Yaskawa INFORM job: DEMO_ROOF_SIDE_0625_3PAINT_57.JBI

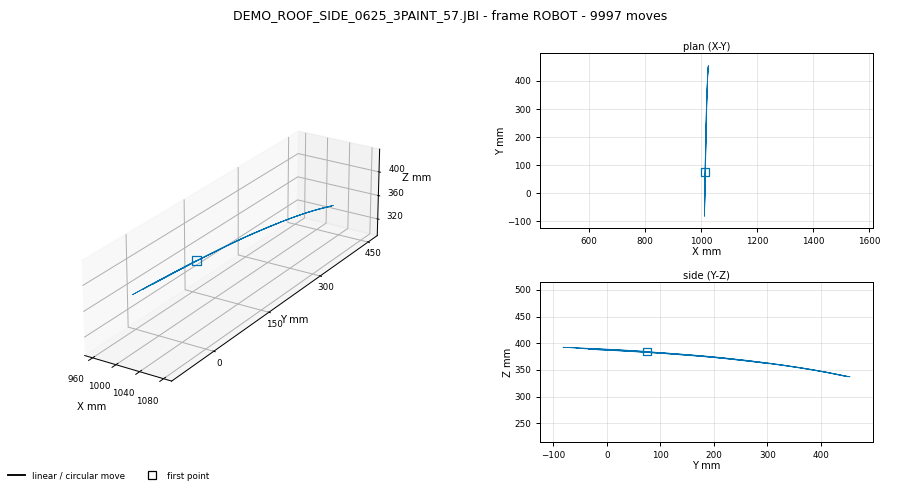
[picture p0: tool path of DEMO_ROOF_SIDE_0625_3PAINT_57.JBI in frame ROBOT, 9997 of 9997 moves have a stored position in this frame; points joined in program order, loops and branches not executed]
/JOB
//NAME DEMO_ROOF_SIDE_0625_3PAINT57
//POS
///NPOS 9997,0,0,0,0,0
///TOOL 0
///USER 0
///POSTYPE ROBOT
///RECTAN
///RCONF 1,0,0,0,0,0,0,0,0,0,0,0,0,0,0,0,0,0,0,0,0,0,0,0
C00000=1015.921,75.710,384.669,166.381,56.145,160.225
C00001=1015.916,75.460,384.686,166.378,56.154,160.227
C00002=1015.911,75.211,384.702,166.376,56.164,160.228
C00003=1015.906,74.930,384.720,166.373,56.174,160.229
C00004=1015.900,74.649,384.737,166.370,56.185,160.231
C00005=1015.894,74.368,384.755,166.367,56.195,160.232
C00006=1015.889,74.087,384.774,166.365,56.207,160.234
C00007=1015.884,73.838,384.789,166.362,56.215,160.235
C00008=1015.879,73.587,384.805,166.358,56.225,160.236
C00009=1015.874,73.339,384.822,166.356,56.235,160.237
C00010=1015.869,73.089,384.837,166.353,56.244,160.238
C00011=1015.864,72.840,384.854,166.351,56.253,160.240
C00012=1015.859,72.590,384.869,166.348,56.263,160.241
C00013=1015.855,72.341,384.885,166.346,56.272,160.242
C00014=1015.849,72.091,384.902,166.344,56.282,160.243
C00015=1015.844,71.842,384.917,166.341,56.291,160.245
C00016=1015.840,71.593,384.933,166.339,56.301,160.246
C00017=1015.834,71.343,384.949,166.336,56.310,160.247
C00018=1015.830,71.093,384.965,166.334,56.319,160.248
C00019=1015.825,70.844,384.981,166.332,56.329,160.250
C00020=1015.820,70.594,384.997,166.328,56.339,160.251
C00021=1015.815,70.345,385.012,166.326,56.348,160.252
C00022=1015.810,70.096,385.028,166.323,56.357,160.253
C00023=1015.806,69.847,385.044,166.320,56.366,160.254
C00024=1015.800,69.597,385.060,166.318,56.376,160.256
C00025=1015.795,69.348,385.076,166.316,56.385,160.257
C00026=1015.790,69.098,385.091,166.313,56.395,160.258
C00027=1015.785,68.848,385.107,166.311,56.404,160.259
C00028=1015.781,68.599,385.124,166.308,56.414,160.261
C00029=1015.776,68.350,385.139,166.306,56.423,160.262
C00030=1015.771,68.100,385.155,166.303,56.432,160.263
C00031=1015.766,67.850,385.170,166.301,56.441,160.264
C00032=1015.761,67.601,385.187,166.298,56.451,160.266
C00033=1015.756,67.352,385.202,166.296,56.460,160.267
C00034=1015.751,67.103,385.217,166.294,56.469,160.268
C00035=1015.746,66.853,385.233,166.290,56.479,160.269
C00036=1015.741,66.603,385.248,166.288,56.489,160.271
C00037=1015.737,66.354,385.264,166.285,56.498,160.272
C00038=1015.731,66.105,385.280,166.283,56.508,160.273
C00039=1015.726,65.855,385.296,166.280,56.516,160.274
C00040=1015.721,65.606,385.311,166.278,56.526,160.275
C00041=1015.716,65.356,385.327,166.275,56.535,160.277
C00042=1015.712,65.107,385.342,166.273,56.545,160.278
C00043=1015.706,64.857,385.358,166.271,56.554,160.279
C00044=1015.701,64.607,385.373,166.268,56.564,160.281
C00045=1015.697,64.359,385.390,166.266,56.573,160.282
C00046=1015.692,64.109,385.405,166.263,56.582,160.283
C00047=1015.686,63.859,385.420,166.261,56.591,160.284
C00048=1015.682,63.610,385.436,166.258,56.601,160.285
C00049=1015.677,63.360,385.451,166.256,56.610,160.287
C00050=1015.672,63.111,385.466,166.253,56.620,160.288
C00051=1015.667,62.862,385.482,166.250,56.630,160.289
C00052=1015.662,62.612,385.498,166.248,56.639,160.290
C00053=1015.657,62.362,385.513,166.245,56.648,160.291
C00054=1015.652,62.113,385.528,166.243,56.658,160.293
C00055=1015.647,61.864,385.543,166.241,56.667,160.294
C00056=1015.642,61.615,385.558,166.238,56.676,160.295
C00057=1015.636,61.364,385.573,166.236,56.686,160.297
C00058=1015.631,61.115,385.588,166.233,56.696,160.298
C00059=1015.626,60.865,385.604,166.230,56.705,160.299
C00060=1015.622,60.616,385.619,166.228,56.715,160.300
C00061=1015.617,60.367,385.635,166.226,56.724,160.302
C00062=1015.611,60.117,385.650,166.223,56.734,160.303
C00063=1015.606,59.867,385.665,166.221,56.743,160.304
C00064=1015.601,59.617,385.680,166.218,56.753,160.305
C00065=1015.596,59.368,385.695,166.215,56.763,160.307
C00066=1015.591,59.119,385.710,166.213,56.772,160.308
C00067=1015.585,58.826,385.728,166.210,56.783,160.309
C00068=1015.579,58.533,385.745,166.207,56.795,160.311
C00069=1015.573,58.240,385.763,166.204,56.805,160.312
C00070=1015.567,57.947,385.782,166.201,56.816,160.314
C00071=1015.563,57.697,385.796,166.199,56.826,160.315
C00072=1015.558,57.447,385.811,166.197,56.835,160.316
C00073=1015.553,57.198,385.826,166.194,56.845,160.317
C00074=1015.547,56.949,385.842,166.191,56.854,160.319
C00075=1015.542,56.700,385.857,166.189,56.864,160.320
C00076=1015.538,56.450,385.871,166.186,56.873,160.321
C00077=1015.533,56.201,385.886,166.184,56.882,160.322
C00078=1015.527,55.951,385.902,166.182,56.892,160.324
C00079=1015.522,55.701,385.917,166.179,56.901,160.325
C00080=1015.517,55.451,385.932,166.177,56.911,160.326
C00081=1015.512,55.202,385.947,166.174,56.920,160.327
C00082=1015.507,54.953,385.962,166.172,56.929,160.328
C00083=1015.503,54.710,385.976,166.170,56.939,160.330
C00084=1015.498,54.466,385.991,166.167,56.948,160.331
C00085=1015.493,54.222,386.006,166.165,56.957,160.332
C00086=1015.488,53.979,386.021,166.162,56.966,160.333
C00087=1015.483,53.735,386.035,166.160,56.975,160.334
C00088=1015.478,53.492,386.050,166.158,56.984,160.336
C00089=1015.473,53.248,386.064,166.156,56.993,160.337
C00090=1015.468,53.004,386.079,166.153,57.002,160.338
C00091=1015.463,52.755,386.094,166.150,57.012,160.339
C00092=1015.458,52.506,386.109,166.148,57.021,160.341
C00093=1015.453,52.256,386.124,166.145,57.030,160.342
C00094=1015.448,52.007,386.139,166.143,57.039,160.343
C00095=1015.443,51.757,386.154,166.141,57.049,160.344
C00096=1015.439,51.508,386.168,166.138,57.058,160.345
C00097=1015.434,51.258,386.184,166.136,57.067,160.347
C00098=1015.428,51.009,386.199,166.134,57.077,160.348
C00099=1015.424,50.759,386.213,166.131,57.086,160.349
C00100=1015.419,50.510,386.228,166.129,57.095,160.350
C00101=1015.414,50.261,386.244,166.126,57.104,160.351
C00102=1015.409,50.011,386.258,166.124,57.114,160.353
C00103=1015.404,49.761,386.273,166.121,57.123,160.354
C00104=1015.399,49.512,386.288,166.119,57.132,160.355
C00105=1015.394,49.262,386.303,166.116,57.142,160.356
C00106=1015.389,49.013,386.318,166.114,57.150,160.357
C00107=1015.384,48.763,386.333,166.112,57.160,160.359
C00108=1015.379,48.514,386.348,166.109,57.169,160.360
C00109=1015.374,48.265,386.363,166.107,57.178,160.361
C00110=1015.369,48.015,386.377,166.104,57.187,160.362
C00111=1015.364,47.766,386.393,166.102,57.197,160.363
C00112=1015.360,47.515,386.408,166.099,57.206,160.364
C00113=1015.355,47.266,386.423,166.098,57.215,160.366
C00114=1015.351,47.016,386.437,166.095,57.224,160.367
C00115=1015.346,46.767,386.452,166.093,57.233,160.368
C00116=1015.341,46.518,386.468,166.090,57.242,160.369
C00117=1015.336,46.268,386.482,166.088,57.252,160.370
C00118=1015.331,46.019,386.497,166.085,57.260,160.371
C00119=1015.327,45.769,386.511,166.083,57.270,160.373
C00120=1015.322,45.520,386.526,166.080,57.279,160.374
C00121=1015.317,45.270,386.541,166.077,57.288,160.375
C00122=1015.312,45.021,386.556,166.075,57.297,160.376
C00123=1015.307,44.771,386.571,166.073,57.306,160.377
C00124=1015.302,44.522,386.586,166.071,57.315,160.379
C00125=1015.297,44.272,386.600,166.069,57.324,160.380
C00126=1015.292,44.023,386.615,166.066,57.333,160.381
C00127=1015.288,43.773,386.630,166.064,57.342,160.382
C00128=1015.282,43.523,386.645,166.061,57.351,160.383
C00129=1015.278,43.274,386.659,166.058,57.360,160.384
C00130=1015.273,43.025,386.674,166.057,57.369,160.386
C00131=1015.267,42.744,386.691,166.054,57.379,160.387
C00132=1015.262,42.463,386.707,166.051,57.389,160.388
C00133=1015.257,42.181,386.724,166.049,57.400,160.390
C00134=1015.251,41.900,386.740,166.046,57.410,160.391
C00135=1015.246,41.651,386.755,166.044,57.419,160.392
C00136=1015.241,41.401,386.770,166.041,57.428,160.393
C00137=1015.236,41.151,386.784,166.039,57.438,160.394
C00138=1015.231,40.902,386.799,166.036,57.447,160.395
C00139=1015.227,40.653,386.813,166.034,57.456,160.397
C00140=1015.221,40.403,386.827,166.031,57.465,160.398
C00141=1015.217,40.153,386.841,166.029,57.474,160.399
C00142=1015.212,39.904,386.856,166.026,57.484,160.400
C00143=1015.207,39.654,386.871,166.024,57.492,160.401
C00144=1015.201,39.405,386.885,166.022,57.502,160.403
C00145=1015.197,39.155,386.899,166.019,57.511,160.404
C00146=1015.192,38.906,386.914,166.017,57.519,160.405
C00147=1015.187,38.657,386.928,166.015,57.529,160.406
C00148=1015.182,38.407,386.942,166.012,57.538,160.407
C00149=1015.177,38.157,386.957,166.010,57.548,160.409
C00150=1015.172,37.908,386.972,166.008,57.556,160.410
C00151=1015.167,37.658,386.986,166.005,57.565,160.411
C00152=1015.163,37.409,387.000,166.003,57.575,160.412
C00153=1015.158,37.159,387.014,166.000,57.584,160.413
C00154=1015.152,36.909,387.028,165.999,57.592,160.414
C00155=1015.147,36.660,387.043,165.996,57.601,160.415
C00156=1015.143,36.410,387.058,165.994,57.611,160.417
C00157=1015.137,36.161,387.072,165.991,57.620,160.418
C00158=1015.133,35.911,387.086,165.989,57.629,160.419
C00159=1015.127,35.662,387.100,165.986,57.638,160.420
C00160=1015.123,35.412,387.114,165.984,57.647,160.421
C00161=1015.117,35.162,387.128,165.982,57.657,160.423
C00162=1015.113,34.913,387.142,165.979,57.666,160.424
C00163=1015.108,34.664,387.156,165.977,57.675,160.425
C00164=1015.103,34.414,387.170,165.974,57.684,160.426
C00165=1015.097,34.164,387.184,165.971,57.693,160.427
C00166=1015.093,33.914,387.199,165.969,57.703,160.428
C00167=1015.088,33.665,387.212,165.967,57.712,160.429
C00168=1015.083,33.416,387.227,165.964,57.720,160.430
C00169=1015.078,33.166,387.240,165.963,57.730,160.432
C00170=1015.073,32.916,387.255,165.960,57.739,160.433
C00171=1015.068,32.667,387.268,165.958,57.747,160.434
C00172=1015.063,32.418,387.282,165.956,57.757,160.435
C00173=1015.058,32.168,387.297,165.953,57.766,160.436
C00174=1015.052,31.918,387.311,165.950,57.775,160.438
C00175=1015.048,31.669,387.325,165.948,57.785,160.439
C00176=1015.043,31.419,387.339,165.946,57.794,160.440
C00177=1015.038,31.170,387.353,165.943,57.802,160.441
C00178=1015.033,30.921,387.367,165.941,57.811,160.442
C00179=1015.028,30.671,387.381,165.939,57.820,160.443
C00180=1015.023,30.421,387.395,165.937,57.829,160.445
C00181=1015.018,30.171,387.409,165.934,57.838,160.446
C00182=1015.014,29.922,387.422,165.931,57.847,160.447
C00183=1015.008,29.672,387.436,165.929,57.856,160.448
C00184=1015.003,29.422,387.450,165.926,57.865,160.449
C00185=1014.998,29.174,387.464,165.925,57.874,160.450
C00186=1014.994,28.924,387.478,165.923,57.883,160.451
C00187=1014.988,28.674,387.492,165.920,57.892,160.453
C00188=1014.984,28.425,387.506,165.917,57.901,160.454
C00189=1014.979,28.175,387.520,165.915,57.910,160.455
C00190=1014.974,27.925,387.535,165.913,57.919,160.456
C00191=1014.969,27.676,387.547,165.911,57.928,160.457
C00192=1014.965,27.426,387.562,165.909,57.937,160.458
C00193=1014.959,27.176,387.576,165.906,57.946,160.459
C00194=1014.954,26.928,387.589,165.903,57.955,160.460
C00195=1014.949,26.646,387.605,165.901,57.965,160.462
C00196=1014.943,26.366,387.620,165.898,57.975,160.463
C00197=1014.937,26.085,387.635,165.895,57.985,160.464
C00198=1014.932,25.804,387.651,165.893,57.996,160.466
C00199=1014.927,25.554,387.664,165.891,58.004,160.467
C00200=1014.922,25.304,387.679,165.889,58.013,160.468
C00201=1014.917,25.055,387.692,165.886,58.022,160.469
C00202=1014.912,24.805,387.706,165.883,58.031,160.470
C00203=1014.906,24.555,387.719,165.881,58.040,160.471
C00204=1014.902,24.306,387.733,165.879,58.050,160.472
C00205=1014.897,24.056,387.746,165.876,58.059,160.474
C00206=1014.892,23.807,387.760,165.875,58.067,160.475
C00207=1014.887,23.557,387.774,165.872,58.076,160.476
C00208=1014.882,23.307,387.787,165.869,58.085,160.477
C00209=1014.877,23.058,387.801,165.867,58.094,160.478
C00210=1014.872,22.808,387.815,165.864,58.103,160.479
C00211=1014.867,22.559,387.828,165.862,58.112,160.480
C00212=1014.862,22.309,387.842,165.860,58.121,160.481
C00213=1014.856,22.060,387.855,165.858,58.130,160.482
C00214=1014.853,21.810,387.869,165.855,58.139,160.484
C00215=1014.847,21.560,387.883,165.853,58.147,160.485
C00216=1014.843,21.311,387.895,165.850,58.156,160.486
C00217=1014.837,21.061,387.909,165.848,58.165,160.487
C00218=1014.832,20.812,387.923,165.846,58.174,160.488
C00219=1014.828,20.562,387.937,165.843,58.183,160.489
C00220=1014.822,20.312,387.950,165.841,58.192,160.490
C00221=1014.818,20.063,387.963,165.839,58.200,160.491
C00222=1014.812,19.813,387.977,165.837,58.209,160.492
C00223=1014.808,19.564,387.990,165.834,58.218,160.494
C00224=1014.803,19.314,388.004,165.832,58.227,160.495
C00225=1014.798,19.065,388.018,165.830,58.236,160.496
C00226=1014.793,18.815,388.031,165.828,58.245,160.497
C00227=1014.788,18.566,388.044,165.825,58.254,160.498
C00228=1014.783,18.316,388.058,165.822,58.263,160.499
C00229=1014.778,18.066,388.070,165.820,58.272,160.500
C00230=1014.773,17.817,388.084,165.818,58.280,160.501
C00231=1014.768,17.567,388.097,165.816,58.289,160.502
C00232=1014.763,17.318,388.111,165.813,58.298,160.504
C00233=1014.758,17.068,388.124,165.811,58.307,160.505
C00234=1014.753,16.818,388.138,165.809,58.315,160.506
C00235=1014.748,16.569,388.150,165.806,58.324,160.507
C00236=1014.743,16.319,388.164,165.804,58.333,160.508
C00237=1014.738,16.070,388.177,165.801,58.342,160.509
C00238=1014.734,15.819,388.191,165.800,58.351,160.510
C00239=1014.729,15.571,388.204,165.797,58.360,160.511
C00240=1014.724,15.320,388.217,165.795,58.369,160.512
C00241=1014.719,15.071,388.230,165.792,58.378,160.513
C00242=1014.714,14.821,388.244,165.790,58.385,160.514
C00243=1014.709,14.572,388.257,165.787,58.394,160.515
C00244=1014.704,14.322,388.270,165.785,58.403,160.516
C00245=1014.699,14.073,388.283,165.784,58.412,160.518
C00246=1014.694,13.822,388.297,165.781,58.421,160.519
C00247=1014.689,13.573,388.309,165.778,58.429,160.520
C00248=1014.684,13.323,388.323,165.776,58.438,160.521
C00249=1014.679,13.074,388.336,165.774,58.447,160.522
C00250=1014.674,12.824,388.349,165.771,58.456,160.523
C00251=1014.669,12.574,388.362,165.769,58.465,160.524
C00252=1014.664,12.326,388.375,165.766,58.474,160.525
C00253=1014.659,12.075,388.388,165.764,58.482,160.526
C00254=1014.654,11.826,388.401,165.762,58.491,160.527
C00255=1014.649,11.576,388.414,165.759,58.500,160.528
C00256=1014.644,11.327,388.426,165.757,58.509,160.529
C00257=1014.638,11.076,388.439,165.755,58.517,160.531
C00258=1014.634,10.827,388.452,165.753,58.526,160.532
C00259=1014.629,10.548,388.467,165.750,58.536,160.533
C00260=1014.622,10.269,388.481,165.748,58.545,160.534
C00261=1014.617,9.989,388.496,165.745,58.556,160.535
C00262=1014.611,9.710,388.509,165.743,58.565,160.537
C00263=1014.606,9.460,388.522,165.740,58.574,160.538
C00264=1014.601,9.210,388.535,165.737,58.583,160.538
C00265=1014.597,8.960,388.548,165.735,58.592,160.540
C00266=1014.590,8.711,388.561,165.733,58.600,160.541
C00267=1014.586,8.462,388.574,165.731,58.609,160.542
C00268=1014.581,8.212,388.587,165.728,58.618,160.543
C00269=1014.576,7.962,388.600,165.725,58.627,160.544
C00270=1014.571,7.713,388.612,165.724,58.635,160.545
C00271=1014.566,7.463,388.625,165.721,58.644,160.546
C00272=1014.561,7.213,388.638,165.718,58.653,160.547
C00273=1014.557,6.964,388.651,165.717,58.661,160.548
C00274=1014.551,6.714,388.663,165.714,58.669,160.549
C00275=1014.546,6.464,388.676,165.711,58.679,160.550
C00276=1014.541,6.215,388.689,165.710,58.687,160.551
C00277=1014.537,5.965,388.702,165.707,58.695,160.552
C00278=1014.531,5.715,388.715,165.704,58.704,160.553
C00279=1014.526,5.466,388.727,165.702,58.712,160.554
C00280=1014.522,5.216,388.740,165.700,58.721,160.555
C00281=1014.517,4.966,388.753,165.699,58.730,160.557
C00282=1014.511,4.717,388.765,165.695,58.738,160.557
C00283=1014.507,4.468,388.778,165.693,58.747,160.558
C00284=1014.502,4.217,388.791,165.691,58.755,160.559
C00285=1014.496,3.968,388.804,165.689,58.764,160.561
C00286=1014.492,3.719,388.816,165.686,58.772,160.561
C00287=1014.487,3.469,388.829,165.684,58.781,160.563
C00288=1014.482,3.219,388.842,165.681,58.789,160.563
C00289=1014.477,2.970,388.854,165.680,58.798,160.565
C00290=1014.472,2.720,388.867,165.677,58.806,160.565
C00291=1014.468,2.471,388.880,165.675,58.815,160.567
C00292=1014.462,2.221,388.893,165.672,58.823,160.568
C00293=1014.457,1.971,388.905,165.669,58.832,160.568
C00294=1014.453,1.722,388.918,165.668,58.840,160.570
C00295=1014.448,1.472,388.931,165.665,58.848,160.570
C00296=1014.443,1.222,388.943,165.663,58.857,160.572
C00297=1014.438,0.972,388.956,165.660,58.865,160.572
C00298=1014.433,0.723,388.968,165.658,58.873,160.573
C00299=1014.429,0.473,388.981,165.656,58.882,160.575
C00300=1014.423,0.224,388.994,165.654,58.890,160.576
C00301=1014.418,-0.026,389.006,165.651,58.899,160.576
C00302=1014.414,-0.275,389.019,165.650,58.907,160.578
C00303=1014.409,-0.525,389.032,165.647,58.916,160.578
C00304=1014.403,-0.775,389.045,165.645,58.923,160.579
C00305=1014.399,-1.025,389.057,165.642,58.932,160.580
C00306=1014.394,-1.274,389.069,165.640,58.940,160.581
C00307=1014.390,-1.524,389.082,165.637,58.949,160.582
C00308=1014.384,-1.773,389.094,165.635,58.957,160.583
C00309=1014.380,-2.023,389.107,165.633,58.964,160.584
C00310=1014.375,-2.273,389.120,165.631,58.974,160.585
C00311=1014.369,-2.522,389.132,165.629,58.981,160.586
C00312=1014.365,-2.772,389.145,165.626,58.990,160.587
C00313=1014.361,-3.022,389.157,165.624,58.998,160.588
C00314=1014.356,-3.271,389.170,165.621,59.006,160.589
C00315=1014.350,-3.521,389.183,165.620,59.015,160.590
C00316=1014.345,-3.770,389.195,165.618,59.022,160.591
C00317=1014.341,-4.021,389.208,165.615,59.031,160.592
C00318=1014.337,-4.270,389.220,165.613,59.039,160.593
C00319=1014.331,-4.519,389.232,165.610,59.047,160.594
C00320=1014.327,-4.769,389.245,165.608,59.055,160.595
C00321=1014.321,-5.019,389.257,165.605,59.064,160.596
C00322=1014.316,-5.268,389.269,165.603,59.072,160.597
C00323=1014.311,-5.546,389.283,165.601,59.081,160.598
C00324=1014.305,-5.823,389.296,165.598,59.091,160.599
C00325=1014.300,-6.101,389.310,165.595,59.100,160.600
C00326=1014.294,-6.377,389.323,165.593,59.109,160.601
C00327=1014.290,-6.628,389.335,165.590,59.118,160.602
C00328=1014.285,-6.877,389.347,165.589,59.126,160.603
C00329=1014.279,-7.126,389.359,165.586,59.134,160.604
C00330=1014.274,-7.377,389.372,165.584,59.142,160.605
C00331=1014.269,-7.626,389.384,165.581,59.150,160.606
C00332=1014.264,-7.876,389.395,165.579,59.159,160.607
C00333=1014.260,-8.125,389.408,165.576,59.167,160.608
C00334=1014.255,-8.375,389.420,165.574,59.175,160.609
C00335=1014.250,-8.625,389.432,165.571,59.184,160.610
C00336=1014.245,-8.874,389.444,165.569,59.192,160.611
C00337=1014.240,-9.124,389.456,165.568,59.199,160.612
C00338=1014.235,-9.374,389.468,165.565,59.208,160.612
C00339=1014.230,-9.623,389.480,165.563,59.217,160.614
C00340=1014.225,-9.873,389.492,165.560,59.225,160.614
C00341=1014.221,-10.123,389.504,165.558,59.233,160.615
C00342=1014.216,-10.372,389.516,165.555,59.241,160.616
C00343=1014.211,-10.622,389.527,165.553,59.249,160.617
C00344=1014.206,-10.871,389.540,165.552,59.257,160.618
C00345=1014.200,-11.122,389.552,165.549,59.265,160.619
C00346=1014.195,-11.371,389.564,165.547,59.273,160.620
C00347=1014.191,-11.621,389.576,165.544,59.282,160.621
C00348=1014.186,-11.871,389.588,165.542,59.290,160.622
C00349=1014.181,-12.120,389.600,165.540,59.298,160.623
C00350=1014.176,-12.370,389.612,165.537,59.306,160.624
C00351=1014.171,-12.619,389.624,165.535,59.314,160.625
C00352=1014.166,-12.869,389.636,165.533,59.322,160.626
C00353=1014.162,-13.119,389.648,165.530,59.330,160.626
C00354=1014.156,-13.368,389.660,165.528,59.337,160.627
C00355=1014.151,-13.618,389.671,165.526,59.345,160.628
C00356=1014.147,-13.868,389.684,165.523,59.354,160.629
C00357=1014.142,-14.117,389.696,165.521,59.362,160.630
C00358=1014.137,-14.367,389.707,165.519,59.369,160.631
C00359=1014.132,-14.617,389.720,165.517,59.377,160.632
C00360=1014.128,-14.866,389.731,165.514,59.386,160.633
C00361=1014.123,-15.116,389.743,165.512,59.393,160.633
C00362=1014.118,-15.365,389.755,165.510,59.401,160.634
C00363=1014.113,-15.615,389.767,165.508,59.409,160.635
C00364=1014.109,-15.865,389.779,165.505,59.417,160.636
C00365=1014.104,-16.115,389.790,165.502,59.424,160.637
C00366=1014.099,-16.364,389.803,165.500,59.432,160.638
C00367=1014.094,-16.614,389.814,165.498,59.441,160.639
C00368=1014.089,-16.864,389.825,165.496,59.449,160.640
C00369=1014.084,-17.113,389.837,165.494,59.457,160.641
C00370=1014.079,-17.363,389.848,165.491,59.465,160.641
C00371=1014.074,-17.613,389.860,165.489,59.473,160.642
C00372=1014.069,-17.863,389.871,165.487,59.481,160.643
C00373=1014.064,-18.113,389.883,165.483,59.489,160.644
C00374=1014.059,-18.362,389.896,165.482,59.497,160.645
C00375=1014.054,-18.612,389.907,165.480,59.505,160.646
C00376=1014.049,-18.862,389.919,165.477,59.513,160.647
C00377=1014.044,-19.112,389.930,165.475,59.521,160.648
C00378=1014.040,-19.361,389.941,165.472,59.528,160.648
C00379=1014.035,-19.610,389.953,165.471,59.536,160.649
C00380=1014.030,-19.860,389.964,165.468,59.544,160.650
C00381=1014.025,-20.110,389.976,165.466,59.552,160.651
C00382=1014.020,-20.360,389.987,165.463,59.560,160.652
C00383=1014.015,-20.610,389.998,165.461,59.568,160.653
C00384=1014.010,-20.859,390.010,165.459,59.576,160.654
C00385=1014.005,-21.109,390.021,165.456,59.583,160.654
C00386=1014.000,-21.358,390.033,165.454,59.591,160.655
C00387=1013.995,-21.634,390.046,165.451,59.600,160.656
C00388=1013.989,-21.909,390.058,165.449,59.609,160.657
C00389=1013.984,-22.185,390.071,165.446,59.617,160.658
C00390=1013.978,-22.460,390.084,165.444,59.625,160.659
C00391=1013.973,-22.710,390.095,165.441,59.633,160.660
C00392=1013.969,-22.960,390.107,165.439,59.641,160.660
C00393=1013.964,-23.210,390.119,165.437,59.649,160.661
C00394=1013.960,-23.459,390.130,165.434,59.656,160.662
C00395=1013.955,-23.709,390.141,165.433,59.664,160.663
C00396=1013.950,-23.958,390.153,165.430,59.671,160.664
C00397=1013.945,-24.208,390.164,165.427,59.680,160.665
C00398=1013.940,-24.458,390.176,165.425,59.687,160.665
C00399=1013.935,-24.707,390.187,165.423,59.695,160.666
C00400=1013.930,-24.957,390.198,165.420,59.702,160.667
C00401=1013.925,-25.207,390.210,165.419,59.710,160.668
C00402=1013.920,-25.457,390.221,165.416,59.717,160.669
C00403=1013.916,-25.706,390.232,165.414,59.725,160.670
C00404=1013.911,-25.956,390.243,165.412,59.732,160.670
C00405=1013.906,-26.206,390.254,165.409,59.740,160.671
C00406=1013.901,-26.456,390.266,165.408,59.748,160.672
C00407=1013.896,-26.706,390.277,165.405,59.755,160.673
C00408=1013.892,-26.955,390.289,165.403,59.762,160.673
C00409=1013.887,-27.204,390.300,165.400,59.770,160.674
C00410=1013.882,-27.454,390.311,165.397,59.778,160.675
C00411=1013.877,-27.704,390.323,165.395,59.785,160.676
C00412=1013.872,-27.953,390.334,165.393,59.793,160.677
C00413=1013.868,-28.204,390.345,165.390,59.800,160.677
C00414=1013.863,-28.453,390.356,165.389,59.808,160.678
C00415=1013.858,-28.703,390.368,165.386,59.815,160.679
C00416=1013.854,-28.953,390.378,165.384,59.823,160.680
C00417=1013.848,-29.202,390.389,165.382,59.831,160.681
C00418=1013.843,-29.452,390.400,165.379,59.838,160.681
C00419=1013.838,-29.701,390.412,165.378,59.846,160.682
C00420=1013.834,-29.952,390.422,165.375,59.853,160.683
C00421=1013.828,-30.201,390.433,165.372,59.861,160.684
C00422=1013.824,-30.450,390.444,165.370,59.869,160.685
C00423=1013.819,-30.701,390.455,165.367,59.876,160.685
C00424=1013.814,-30.950,390.467,165.365,59.883,160.686
C00425=1013.808,-31.200,390.477,165.362,59.890,160.687
C00426=1013.804,-31.450,390.488,165.361,59.898,160.688
C00427=1013.799,-31.699,390.499,165.358,59.906,160.688
C00428=1013.795,-31.949,390.510,165.356,59.913,160.689
C00429=1013.789,-32.199,390.521,165.353,59.920,160.690
C00430=1013.784,-32.448,390.532,165.351,59.928,160.691
C00431=1013.780,-32.698,390.542,165.349,59.935,160.691
C00432=1013.775,-32.948,390.554,165.347,59.943,160.692
C00433=1013.769,-33.197,390.565,165.344,59.950,160.693
C00434=1013.765,-33.447,390.575,165.342,59.957,160.693
C00435=1013.760,-33.697,390.587,165.340,59.965,160.694
C00436=1013.756,-33.947,390.597,165.337,59.972,160.695
C00437=1013.751,-34.196,390.608,165.335,59.980,160.696
C00438=1013.746,-34.447,390.619,165.333,59.987,160.697
C00439=1013.741,-34.696,390.630,165.331,59.994,160.697
C00440=1013.736,-34.946,390.641,165.329,60.001,160.698
C00441=1013.731,-35.196,390.651,165.326,60.008,160.699
C00442=1013.727,-35.445,390.663,165.324,60.016,160.699
C00443=1013.722,-35.695,390.673,165.321,60.023,160.700
C00444=1013.717,-35.944,390.684,165.319,60.030,160.701
C00445=1013.712,-36.194,390.695,165.317,60.037,160.702
C00446=1013.707,-36.444,390.706,165.314,60.045,160.702
C00447=1013.703,-36.694,390.716,165.312,60.052,160.703
C00448=1013.698,-36.944,390.728,165.310,60.059,160.704
C00449=1013.693,-37.193,390.738,165.308,60.066,160.704
C00450=1013.688,-37.443,390.749,165.305,60.073,160.705
C00451=1013.683,-37.717,390.761,165.303,60.080,160.706
C00452=1013.678,-37.991,390.773,165.300,60.089,160.707
C00453=1013.673,-38.266,390.785,165.298,60.096,160.707
C00454=1013.668,-38.540,390.797,165.295,60.105,160.708
C00455=1013.662,-38.791,390.807,165.294,60.111,160.709
C00456=1013.658,-39.040,390.818,165.290,60.118,160.709
C00457=1013.653,-39.290,390.829,165.288,60.125,160.710
C00458=1013.648,-39.539,390.839,165.286,60.133,160.711
C00459=1013.643,-39.789,390.850,165.284,60.139,160.712
C00460=1013.639,-40.039,390.861,165.282,60.147,160.712
C00461=1013.634,-40.289,390.871,165.279,60.154,160.713
C00462=1013.629,-40.538,390.882,165.277,60.161,160.714
C00463=1013.624,-40.788,390.892,165.275,60.168,160.714
C00464=1013.619,-41.038,390.902,165.271,60.175,160.715
C00465=1013.614,-41.288,390.913,165.270,60.182,160.716
C00466=1013.609,-41.537,390.923,165.268,60.189,160.716
C00467=1013.605,-41.787,390.934,165.265,60.196,160.717
C00468=1013.600,-42.037,390.944,165.263,60.204,160.718
C00469=1013.595,-42.287,390.955,165.260,60.211,160.718
C00470=1013.590,-42.536,390.965,165.258,60.217,160.719
C00471=1013.586,-42.786,390.976,165.256,60.224,160.720
C00472=1013.580,-43.036,390.986,165.254,60.232,160.720
C00473=1013.576,-43.285,390.996,165.251,60.239,160.721
C00474=1013.571,-43.536,391.006,165.249,60.245,160.722
C00475=1013.566,-43.785,391.017,165.247,60.252,160.722
C00476=1013.561,-44.035,391.028,165.244,60.259,160.723
C00477=1013.557,-44.285,391.038,165.241,60.266,160.723
C00478=1013.552,-44.534,391.048,165.240,60.273,160.724
C00479=1013.547,-44.784,391.058,165.238,60.280,160.725
C00480=1013.542,-45.033,391.069,165.234,60.287,160.725
C00481=1013.537,-45.283,391.079,165.233,60.293,160.726
C00482=1013.533,-45.533,391.090,165.231,60.301,160.727
C00483=1013.527,-45.783,391.100,165.228,60.307,160.727
C00484=1013.523,-46.033,391.110,165.226,60.314,160.728
C00485=1013.518,-46.282,391.120,165.223,60.321,160.728
C00486=1013.514,-46.533,391.131,165.221,60.328,160.729
C00487=1013.509,-46.781,391.141,165.219,60.334,160.730
C00488=1013.504,-47.031,391.152,165.216,60.341,160.730
C00489=1013.499,-47.281,391.162,165.214,60.347,160.731
C00490=1013.495,-47.531,391.172,165.212,60.355,160.732
C00491=1013.490,-47.781,391.182,165.209,60.361,160.732
C00492=1013.485,-48.030,391.192,165.208,60.368,160.733
C00493=1013.481,-48.280,391.202,165.205,60.375,160.733
C00494=1013.475,-48.530,391.213,165.203,60.381,160.734
C00495=1013.471,-48.780,391.223,165.200,60.388,160.734
C00496=1013.466,-49.029,391.233,165.198,60.394,160.735
C00497=1013.461,-49.279,391.244,165.196,60.401,160.736
C00498=1013.456,-49.529,391.254,165.194,60.407,160.736
C00499=1013.452,-49.778,391.264,165.191,60.415,160.737
C00500=1013.447,-50.028,391.275,165.189,60.421,160.738
C00501=1013.443,-50.278,391.285,165.186,60.427,160.738
C00502=1013.438,-50.528,391.295,165.185,60.434,160.739
C00503=1013.433,-50.778,391.306,165.182,60.441,160.739
C00504=1013.428,-51.027,391.315,165.180,60.447,160.740
C00505=1013.424,-51.277,391.326,165.177,60.453,160.740
C00506=1013.419,-51.528,391.335,165.176,60.460,160.741
C00507=1013.414,-51.777,391.345,165.173,60.467,160.741
C00508=1013.410,-52.027,391.355,165.170,60.474,160.742
C00509=1013.404,-52.277,391.365,165.168,60.480,160.743
C00510=1013.400,-52.527,391.374,165.166,60.488,160.743
C00511=1013.395,-52.776,391.384,165.164,60.494,160.744
C00512=1013.390,-53.026,391.394,165.161,60.500,160.744
C00513=1013.384,-53.276,391.404,165.160,60.507,160.745
C00514=1013.380,-53.526,391.413,165.157,60.514,160.745
C00515=1013.375,-53.800,391.423,165.154,60.521,160.746
C00516=1013.369,-54.075,391.434,165.152,60.528,160.747
C00517=1013.363,-54.350,391.445,165.149,60.536,160.747
C00518=1013.358,-54.624,391.455,165.147,60.543,160.748
C00519=1013.354,-54.874,391.466,165.144,60.549,160.749
C00520=1013.349,-55.124,391.476,165.142,60.556,160.749
C00521=1013.344,-55.374,391.485,165.139,60.562,160.749
C00522=1013.340,-55.623,391.495,165.138,60.569,160.750
C00523=1013.335,-55.872,391.505,165.135,60.576,160.751
C00524=1013.330,-56.123,391.514,165.133,60.582,160.751
C00525=1013.325,-56.373,391.524,165.131,60.588,160.752
C00526=1013.320,-56.622,391.534,165.128,60.594,160.752
C00527=1013.315,-56.872,391.543,165.126,60.600,160.753
C00528=1013.311,-57.121,391.552,165.123,60.608,160.753
C00529=1013.306,-57.371,391.562,165.121,60.614,160.754
C00530=1013.301,-57.622,391.572,165.119,60.620,160.755
C00531=1013.296,-57.871,391.581,165.116,60.627,160.755
C00532=1013.291,-58.121,391.591,165.114,60.633,160.755
C00533=1013.286,-58.370,391.600,165.111,60.639,160.756
C00534=1013.282,-58.620,391.610,165.109,60.645,160.756
C00535=1013.277,-58.870,391.619,165.107,60.651,160.757
C00536=1013.272,-59.120,391.629,165.104,60.658,160.757
C00537=1013.267,-59.370,391.638,165.102,60.664,160.758
C00538=1013.262,-59.619,391.648,165.100,60.670,160.758
C00539=1013.257,-59.869,391.658,165.098,60.676,160.759
C00540=1013.253,-60.119,391.667,165.095,60.683,160.759
C00541=1013.248,-60.368,391.677,165.093,60.689,160.760
C00542=1013.244,-60.618,391.686,165.092,60.695,160.760
C00543=1013.239,-60.868,391.696,165.090,60.701,160.761
C00544=1013.234,-61.118,391.705,165.086,60.707,160.761
C00545=1013.229,-61.368,391.716,165.084,60.713,160.762
C00546=1013.225,-61.618,391.725,165.082,60.719,160.762
C00547=1013.220,-61.868,391.735,165.080,60.725,160.763
C00548=1013.215,-62.117,391.744,165.077,60.732,160.763
C00549=1013.211,-62.367,391.753,165.075,60.738,160.764
C00550=1013.206,-62.616,391.763,165.072,60.744,160.764
C00551=1013.201,-62.866,391.772,165.070,60.750,160.764
C00552=1013.197,-63.116,391.782,165.068,60.756,160.765
C00553=1013.192,-63.366,391.791,165.066,60.761,160.765
C00554=1013.187,-63.615,391.801,165.064,60.767,160.766
C00555=1013.183,-63.865,391.810,165.061,60.774,160.766
C00556=1013.178,-64.115,391.820,165.059,60.780,160.767
C00557=1013.173,-64.365,391.829,165.056,60.785,160.767
C00558=1013.169,-64.615,391.838,165.054,60.791,160.767
C00559=1013.164,-64.864,391.848,165.052,60.797,160.768
C00560=1013.159,-65.114,391.857,165.050,60.803,160.768
///RCONF 1,0,0,0,1,0,0,0,0,0,0,0,0,0,0,0,0,0,0,0,0,0,0,0
C00561=1013.155,-65.364,391.867,165.048,60.809,160.769
C00562=1013.150,-65.614,391.876,165.045,60.814,160.769
C00563=1013.145,-65.863,391.886,165.043,60.821,160.770
C00564=1013.141,-66.113,391.895,165.040,60.826,160.770
C00565=1013.136,-66.362,391.904,165.039,60.832,160.770
C00566=1013.131,-66.613,391.913,165.036,60.837,160.771
C00567=1013.127,-66.863,391.923,165.034,60.844,160.771
C00568=1013.122,-67.112,391.932,165.031,60.849,160.771
C00569=1013.117,-67.362,391.941,165.029,60.855,160.772
C00570=1013.113,-67.611,391.951,165.027,60.860,160.772
C00571=1013.108,-67.861,391.960,165.025,60.867,160.773
C00572=1013.104,-68.111,391.969,165.022,60.872,160.773
C00573=1013.099,-68.361,391.979,165.020,60.877,160.773
C00574=1013.094,-68.611,391.988,165.018,60.883,160.774
C00575=1013.090,-68.861,391.997,165.015,60.889,160.774
C00576=1013.085,-69.110,392.007,165.012,60.894,160.774
C00577=1013.080,-69.360,392.016,165.010,60.900,160.775
C00578=1013.076,-69.610,392.025,165.009,60.905,160.775
C00579=1013.068,-70.020,392.041,165.005,60.914,160.776
C00580=1013.061,-70.430,392.056,165.001,60.923,160.776
C00581=1013.053,-70.840,392.071,164.997,60.932,160.777
C00582=1013.046,-71.250,392.086,164.994,60.941,160.777
C00583=1013.041,-71.499,392.096,164.991,60.947,160.778
C00584=1013.037,-71.749,392.105,164.988,60.952,160.778
C00585=1013.032,-71.999,392.114,164.986,60.958,160.778
C00586=1013.027,-72.249,392.124,164.985,60.963,160.779
C00587=1013.023,-72.499,392.133,164.982,60.969,160.779
C00588=1013.018,-72.749,392.142,164.980,60.974,160.779
C00589=1013.014,-72.999,392.151,164.977,60.979,160.779
C00590=1013.009,-73.248,392.161,164.975,60.984,160.780
C00591=1013.005,-73.498,392.170,164.973,60.990,160.780
C00592=1013.001,-73.748,392.179,164.970,60.995,160.780
C00593=1012.996,-73.998,392.188,164.969,61.000,160.781
C00594=1012.991,-74.247,392.198,164.966,61.005,160.781
C00595=1012.987,-74.497,392.207,164.963,61.011,160.781
C00596=1012.982,-74.747,392.216,164.962,61.016,160.782
C00597=1012.978,-74.997,392.225,164.959,61.021,160.782
C00598=1012.974,-75.246,392.234,164.957,61.026,160.782
C00599=1012.968,-75.496,392.242,164.954,61.032,160.782
C00600=1012.964,-75.746,392.251,164.952,61.037,160.783
C00601=1012.959,-75.996,392.260,164.950,61.042,160.783
C00602=1012.955,-76.246,392.269,164.948,61.048,160.783
C00603=1012.950,-76.495,392.277,164.946,61.053,160.784
C00604=1012.946,-76.745,392.287,164.944,61.059,160.784
C00605=1012.941,-76.995,392.296,164.941,61.064,160.784
C00606=1012.936,-77.245,392.304,164.938,61.069,160.784
C00607=1012.931,-77.495,392.313,164.936,61.074,160.785
C00608=1012.927,-77.744,392.322,164.934,61.079,160.785
C00609=1012.922,-77.994,392.330,164.932,61.084,160.785
C00610=1012.918,-78.244,392.339,164.929,61.089,160.785
C00611=1012.913,-78.494,392.349,164.927,61.095,160.786
C00612=1012.909,-78.743,392.357,164.925,61.100,160.786
C00613=1012.904,-78.993,392.366,164.923,61.105,160.786
C00614=1012.899,-79.243,392.375,164.921,61.110,160.787
C00615=1012.895,-79.493,392.384,164.918,61.115,160.787
C00616=1012.890,-79.742,392.392,164.915,61.120,160.787
C00617=1012.886,-79.993,392.400,164.914,61.125,160.787
C00618=1012.882,-80.243,392.409,164.911,61.130,160.787
C00619=1012.877,-80.493,392.419,164.909,61.135,160.788
C00620=1012.872,-80.742,392.427,164.906,61.140,160.788
C00621=1012.867,-80.992,392.435,164.905,61.145,160.788
C00622=1012.863,-81.242,392.444,164.902,61.150,160.788
C00623=1012.858,-81.492,392.452,164.900,61.155,160.789
C00624=1012.854,-81.741,392.461,164.898,61.160,160.789
C00625=1012.848,-81.991,392.469,164.894,61.165,160.789
C00626=1012.844,-82.242,392.478,164.893,61.170,160.789
C00627=1012.844,-69.994,391.617,164.988,61.168,160.820
C00628=1012.851,-69.639,391.604,164.992,61.161,160.820
C00629=1012.855,-69.390,391.594,164.994,61.156,160.820
C00630=1012.860,-69.140,391.585,164.996,61.151,160.819
C00631=1012.864,-68.890,391.576,164.999,61.145,160.819
C00632=1012.869,-68.640,391.566,165.000,61.140,160.819
C00633=1012.874,-68.390,391.557,165.003,61.135,160.818
C00634=1012.878,-68.140,391.548,165.006,61.130,160.818
C00635=1012.883,-67.891,391.538,165.007,61.125,160.818
C00636=1012.888,-67.641,391.529,165.010,61.119,160.818
C00637=1012.892,-67.391,391.520,165.012,61.114,160.817
C00638=1012.897,-67.141,391.510,165.014,61.109,160.817
C00639=1012.902,-66.891,391.501,165.016,61.103,160.816
C00640=1012.906,-66.641,391.492,165.018,61.097,160.816
C00641=1012.911,-66.392,391.482,165.021,61.092,160.816
C00642=1012.915,-66.142,391.473,165.023,61.087,160.815
C00643=1012.920,-65.892,391.464,165.025,61.082,160.815
C00644=1012.925,-65.642,391.455,165.028,61.076,160.815
C00645=1012.929,-65.392,391.445,165.030,61.070,160.814
C00646=1012.934,-65.143,391.436,165.032,61.065,160.814
C00647=1012.939,-64.893,391.427,165.034,61.060,160.814
C00648=1012.944,-64.644,391.417,165.036,61.054,160.813
C00649=1012.948,-64.394,391.408,165.038,61.048,160.813
C00650=1012.953,-64.143,391.399,165.041,61.043,160.813
///RCONF 1,0,0,0,0,0,0,0,0,0,0,0,0,0,0,0,0,0,0,0,0,0,0,0
C00651=1012.957,-63.894,391.389,165.044,61.038,160.812
C00652=1012.962,-63.644,391.380,165.045,61.031,160.812
C00653=1012.967,-63.395,391.370,165.048,61.026,160.812
C00654=1012.971,-63.145,391.361,165.050,61.021,160.811
C00655=1012.976,-62.895,391.351,165.052,61.015,160.811
C00656=1012.981,-62.645,391.342,165.054,61.010,160.810
C00657=1012.985,-62.396,391.332,165.056,61.003,160.810
C00658=1012.990,-62.146,391.323,165.059,60.998,160.810
C00659=1012.995,-61.896,391.313,165.061,60.993,160.809
C00660=1012.999,-61.646,391.304,165.063,60.987,160.809
C00661=1013.004,-61.397,391.294,165.066,60.981,160.809
C00662=1013.009,-61.147,391.285,165.068,60.975,160.808
C00663=1013.014,-60.897,391.276,165.070,60.970,160.808
C00664=1013.018,-60.647,391.267,165.072,60.964,160.807
C00665=1013.022,-60.398,391.256,165.074,60.957,160.807
C00666=1013.027,-60.148,391.247,165.077,60.952,160.806
C00667=1013.032,-59.898,391.237,165.079,60.946,160.806
C00668=1013.036,-59.648,391.228,165.081,60.940,160.806
C00669=1013.041,-59.398,391.218,165.083,60.934,160.805
C00670=1013.046,-59.148,391.209,165.085,60.928,160.804
C00671=1013.051,-58.899,391.199,165.088,60.923,160.804
C00672=1013.055,-58.649,391.190,165.090,60.917,160.804
C00673=1013.060,-58.399,391.180,165.093,60.910,160.803
C00674=1013.065,-58.150,391.170,165.095,60.905,160.803
C00675=1013.070,-57.900,391.161,165.097,60.899,160.802
C00676=1013.074,-57.650,391.152,165.099,60.892,160.802
C00677=1013.079,-57.400,391.142,165.101,60.886,160.801
C00678=1013.084,-57.150,391.132,165.104,60.881,160.801
C00679=1013.089,-56.901,391.123,165.106,60.875,160.800
C00680=1013.094,-56.651,391.113,165.109,60.868,160.800
C00681=1013.099,-56.401,391.104,165.111,60.862,160.800
C00682=1013.103,-56.151,391.095,165.112,60.856,160.799
C00683=1013.108,-55.902,391.085,165.114,60.850,160.798
C00684=1013.113,-55.652,391.075,165.117,60.845,160.798
C00685=1013.118,-55.402,391.066,165.120,60.838,160.798
C00686=1013.123,-55.152,391.056,165.122,60.832,160.797
C00687=1013.128,-54.903,391.046,165.124,60.826,160.797
C00688=1013.132,-54.653,391.037,165.126,60.820,160.796
C00689=1013.138,-54.378,391.026,165.128,60.812,160.795
C00690=1013.142,-54.104,391.015,165.131,60.806,160.795
C00691=1013.147,-53.830,391.005,165.133,60.798,160.794
C00692=1013.153,-53.555,390.994,165.137,60.792,160.794
C00693=1013.158,-53.305,390.984,165.138,60.786,160.793
C00694=1013.163,-53.056,390.974,165.140,60.779,160.793
C00695=1013.168,-52.805,390.965,165.143,60.773,160.792
C00696=1013.172,-52.556,390.955,165.145,60.766,160.791
C00697=1013.177,-52.306,390.945,165.148,60.759,160.791
C00698=1013.182,-52.056,390.936,165.150,60.753,160.791
C00699=1013.187,-51.807,390.926,165.152,60.747,160.790
C00700=1013.192,-51.557,390.916,165.155,60.741,160.790
C00701=1013.197,-51.307,390.906,165.156,60.734,160.789
C00702=1013.201,-51.057,390.897,165.158,60.728,160.788
C00703=1013.206,-50.807,390.887,165.161,60.722,160.788
C00704=1013.210,-50.557,390.876,165.163,60.716,160.788
C00705=1013.215,-50.308,390.866,165.165,60.710,160.787
C00706=1013.220,-50.057,390.856,165.167,60.703,160.786
C00707=1013.225,-49.808,390.846,165.170,60.697,160.786
C00708=1013.229,-49.559,390.836,165.172,60.691,160.785
C00709=1013.234,-49.309,390.826,165.174,60.685,160.785
C00710=1013.239,-49.059,390.815,165.177,60.677,160.784
C00711=1013.243,-48.809,390.805,165.178,60.671,160.784
C00712=1013.248,-48.560,390.795,165.180,60.665,160.783
C00713=1013.253,-48.309,390.785,165.183,60.659,160.783
C00714=1013.257,-48.060,390.775,165.185,60.652,160.782
C00715=1013.262,-47.810,390.764,165.188,60.646,160.782
C00716=1013.267,-47.561,390.753,165.190,60.640,160.781
C00717=1013.271,-47.311,390.743,165.192,60.633,160.780
C00718=1013.276,-47.061,390.733,165.195,60.626,160.780
C00719=1013.282,-46.811,390.723,165.197,60.620,160.779
C00720=1013.286,-46.562,390.713,165.200,60.614,160.779
C00721=1013.291,-46.312,390.703,165.201,60.607,160.778
C00722=1013.295,-46.062,390.692,165.204,60.600,160.778
C00723=1013.300,-45.812,390.682,165.206,60.594,160.777
C00724=1013.304,-45.563,390.672,165.208,60.587,160.776
C00725=1013.310,-45.313,390.662,165.210,60.581,160.776
C00726=1013.314,-45.063,390.651,165.212,60.575,160.775
C00727=1013.319,-44.814,390.641,165.215,60.567,160.774
C00728=1013.324,-44.564,390.630,165.218,60.561,160.774
C00729=1013.328,-44.314,390.620,165.220,60.555,160.774
C00730=1013.333,-44.064,390.610,165.222,60.547,160.773
C00731=1013.338,-43.814,390.600,165.224,60.541,160.772
C00732=1013.342,-43.565,390.589,165.226,60.534,160.772
C00733=1013.347,-43.315,390.579,165.228,60.528,160.771
C00734=1013.353,-43.066,390.569,165.231,60.520,160.770
C00735=1013.357,-42.815,390.558,165.232,60.514,160.770
C00736=1013.362,-42.566,390.548,165.235,60.507,160.769
C00737=1013.366,-42.316,390.538,165.238,60.501,160.769
C00738=1013.372,-42.066,390.528,165.239,60.494,160.768
C00739=1013.376,-41.816,390.517,165.242,60.487,160.767
C00740=1013.381,-41.567,390.506,165.243,60.480,160.766
C00741=1013.386,-41.317,390.496,165.246,60.473,160.766
C00742=1013.391,-41.067,390.486,165.249,60.466,160.765
C00743=1013.395,-40.817,390.475,165.250,60.460,160.764
C00744=1013.401,-40.568,390.465,165.253,60.452,160.764
C00745=1013.405,-40.318,390.454,165.256,60.446,160.763
C00746=1013.410,-40.069,390.444,165.257,60.439,160.762
C00747=1013.414,-39.818,390.434,165.259,60.432,160.762
C00748=1013.419,-39.569,390.424,165.262,60.425,160.761
C00749=1013.424,-39.319,390.412,165.264,60.418,160.760
C00750=1013.428,-39.069,390.402,165.267,60.412,160.760
C00751=1013.434,-38.820,390.391,165.269,60.404,160.759
C00752=1013.438,-38.570,390.381,165.270,60.398,160.758
C00753=1013.443,-38.296,390.369,165.274,60.390,160.758
C00754=1013.449,-38.021,390.356,165.276,60.382,160.757
C00755=1013.454,-37.748,390.345,165.279,60.375,160.757
C00756=1013.459,-37.473,390.333,165.281,60.368,160.756
C00757=1013.463,-37.223,390.323,165.283,60.361,160.755
C00758=1013.468,-36.974,390.311,165.286,60.353,160.755
C00759=1013.473,-36.724,390.302,165.287,60.346,160.754
C00760=1013.478,-36.474,390.290,165.290,60.340,160.753
C00761=1013.482,-36.225,390.280,165.292,60.333,160.753
C00762=1013.487,-35.975,390.268,165.294,60.326,160.752
C00763=1013.493,-35.725,390.258,165.296,60.319,160.751
C00764=1013.497,-35.476,390.247,165.299,60.312,160.751
C00765=1013.502,-35.225,390.236,165.302,60.305,160.750
C00766=1013.506,-34.976,390.225,165.303,60.298,160.749
C00767=1013.512,-34.726,390.215,165.305,60.291,160.748
C00768=1013.516,-34.477,390.204,165.308,60.283,160.748
C00769=1013.521,-34.226,390.193,165.310,60.276,160.747
C00770=1013.526,-33.977,390.182,165.312,60.269,160.746
C00771=1013.531,-33.727,390.172,165.314,60.263,160.746
C00772=1013.536,-33.477,390.160,165.317,60.255,160.745
C00773=1013.540,-33.228,390.150,165.319,60.248,160.744
C00774=1013.545,-32.978,390.139,165.322,60.241,160.743
C00775=1013.550,-32.729,390.128,165.324,60.234,160.743
C00776=1013.555,-32.479,390.117,165.326,60.226,160.742
C00777=1013.560,-32.229,390.106,165.328,60.219,160.741
C00778=1013.564,-31.979,390.095,165.330,60.212,160.740
C00779=1013.569,-31.730,390.084,165.333,60.205,160.740
C00780=1013.574,-31.479,390.074,165.335,60.198,160.739
C00781=1013.579,-31.230,390.063,165.337,60.190,160.738
C00782=1013.584,-30.980,390.051,165.340,60.183,160.738
C00783=1013.588,-30.731,390.041,165.341,60.175,160.737
C00784=1013.593,-30.481,390.030,165.344,60.168,160.736
C00785=1013.598,-30.231,390.019,165.346,60.160,160.735
C00786=1013.602,-29.982,390.008,165.349,60.153,160.734
C00787=1013.607,-29.732,389.997,165.351,60.146,160.734
C00788=1013.613,-29.482,389.986,165.354,60.139,160.733
C00789=1013.617,-29.233,389.975,165.356,60.131,160.732
C00790=1013.622,-28.983,389.964,165.358,60.123,160.731
C00791=1013.627,-28.732,389.953,165.360,60.116,160.731
C00792=1013.632,-28.484,389.943,165.362,60.109,160.730
C00793=1013.637,-28.234,389.931,165.365,60.102,160.729
C00794=1013.642,-27.983,389.920,165.367,60.094,160.728
C00795=1013.646,-27.734,389.909,165.368,60.087,160.727
C00796=1013.651,-27.484,389.898,165.370,60.079,160.727
C00797=1013.656,-27.235,389.886,165.373,60.072,160.726
C00798=1013.661,-26.984,389.876,165.375,60.065,160.725
C00799=1013.665,-26.735,389.864,165.378,60.058,160.725
C00800=1013.670,-26.485,389.853,165.379,60.050,160.723
C00801=1013.675,-26.236,389.841,165.382,60.042,160.723
C00802=1013.680,-25.986,389.830,165.384,60.035,160.722
C00803=1013.685,-25.737,389.819,165.387,60.028,160.721
C00804=1013.690,-25.487,389.807,165.389,60.021,160.721
C00805=1013.695,-25.237,389.796,165.391,60.013,160.720
C00806=1013.699,-24.988,389.785,165.393,60.005,160.719
C00807=1013.704,-24.738,389.774,165.396,59.998,160.718
C00808=1013.708,-24.487,389.762,165.398,59.991,160.718
C00809=1013.713,-24.238,389.751,165.400,59.983,160.717
C00810=1013.717,-23.989,389.739,165.402,59.976,160.716
C00811=1013.722,-23.739,389.728,165.405,59.968,160.715
C00812=1013.727,-23.489,389.716,165.407,59.960,160.714
C00813=1013.732,-23.239,389.705,165.409,59.953,160.713
C00814=1013.737,-22.990,389.694,165.411,59.946,160.713
C00815=1013.742,-22.740,389.682,165.413,59.938,160.712
C00816=1013.747,-22.490,389.671,165.416,59.931,160.711
C00817=1013.753,-22.215,389.659,165.419,59.922,160.710
C00818=1013.758,-21.940,389.645,165.421,59.914,160.709
C00819=1013.763,-21.664,389.634,165.422,59.905,160.708
C00820=1013.768,-21.389,389.621,165.425,59.897,160.707
C00821=1013.773,-21.139,389.610,165.428,59.889,160.706
C00822=1013.778,-20.889,389.598,165.430,59.881,160.705
C00823=1013.783,-20.639,389.587,165.433,59.874,160.705
C00824=1013.787,-20.390,389.575,165.435,59.866,160.704
C00825=1013.792,-20.141,389.564,165.437,59.858,160.703
C00826=1013.797,-19.891,389.553,165.439,59.850,160.702
C00827=1013.802,-19.641,389.541,165.442,59.843,160.702
C00828=1013.807,-19.391,389.530,165.443,59.835,160.700
C00829=1013.812,-19.142,389.518,165.446,59.827,160.700
C00830=1013.817,-18.892,389.507,165.449,59.819,160.699
C00831=1013.822,-18.642,389.496,165.450,59.812,160.698
C00832=1013.827,-18.393,389.483,165.452,59.804,160.697
C00833=1013.831,-18.143,389.471,165.455,59.796,160.696
C00834=1013.836,-17.893,389.460,165.458,59.788,160.695
C00835=1013.841,-17.644,389.448,165.459,59.780,160.694
C00836=1013.846,-17.394,389.437,165.462,59.773,160.694
C00837=1013.851,-17.145,389.426,165.464,59.765,160.693
C00838=1013.856,-16.895,389.414,165.467,59.756,160.692
C00839=1013.861,-16.645,389.403,165.468,59.748,160.691
C00840=1013.866,-16.395,389.391,165.471,59.741,160.690
C00841=1013.871,-16.145,389.380,165.474,59.733,160.689
C00842=1013.875,-15.895,389.368,165.476,59.725,160.688
C00843=1013.880,-15.646,389.356,165.478,59.717,160.688
C00844=1013.885,-15.396,389.344,165.480,59.709,160.687
C00845=1013.890,-15.146,389.332,165.482,59.701,160.686
C00846=1013.895,-14.896,389.321,165.484,59.694,160.685
C00847=1013.900,-14.647,389.308,165.487,59.686,160.684
C00848=1013.904,-14.397,389.296,165.489,59.678,160.683
C00849=1013.909,-14.147,389.285,165.491,59.671,160.682
C00850=1013.914,-13.899,389.273,165.493,59.663,160.681
C00851=1013.918,-13.649,389.261,165.496,59.654,160.681
C00852=1013.923,-13.399,389.250,165.498,59.646,160.680
C00853=1013.928,-13.150,389.237,165.500,59.639,160.679
C00854=1013.933,-12.900,389.225,165.502,59.631,160.678
C00855=1013.938,-12.650,389.214,165.505,59.623,160.677
C00856=1013.943,-12.401,389.202,165.507,59.615,160.676
C00857=1013.947,-12.151,389.190,165.509,59.607,160.675
C00858=1013.952,-11.901,389.178,165.511,59.600,160.674
C00859=1013.958,-11.652,389.166,165.514,59.591,160.673
C00860=1013.962,-11.401,389.154,165.516,59.583,160.672
C00861=1013.967,-11.152,389.142,165.518,59.575,160.671
C00862=1013.972,-10.902,389.130,165.521,59.567,160.671
C00863=1013.976,-10.652,389.118,165.523,59.559,160.670
C00864=1013.981,-10.403,389.107,165.524,59.551,160.669
C00865=1013.987,-10.153,389.094,165.527,59.543,160.668
C00866=1013.991,-9.903,389.082,165.529,59.535,160.667
C00867=1013.996,-9.654,389.070,165.531,59.527,160.666
C00868=1014.001,-9.404,389.059,165.534,59.518,160.665
C00869=1014.006,-9.155,389.046,165.536,59.510,160.664
C00870=1014.011,-8.905,389.034,165.539,59.502,160.663
C00871=1014.016,-8.655,389.023,165.541,59.494,160.662
C00872=1014.020,-8.406,389.010,165.542,59.486,160.661
C00873=1014.025,-8.156,388.999,165.545,59.478,160.660
C00874=1014.030,-7.906,388.986,165.547,59.470,160.659
C00875=1014.035,-7.657,388.974,165.550,59.461,160.658
C00876=1014.040,-7.407,388.962,165.552,59.453,160.657
C00877=1014.045,-7.157,388.950,165.554,59.445,160.656
C00878=1014.050,-6.907,388.939,165.557,59.437,160.656
C00879=1014.055,-6.658,388.927,165.559,59.429,160.655
C00880=1014.060,-6.407,388.914,165.562,59.421,160.654
C00881=1014.065,-6.131,388.901,165.564,59.412,160.653
C00882=1014.071,-5.854,388.888,165.566,59.402,160.652
C00883=1014.076,-5.577,388.874,165.568,59.393,160.650
C00884=1014.082,-5.300,388.861,165.572,59.384,160.649
C00885=1014.086,-5.050,388.849,165.574,59.376,160.648
C00886=1014.091,-4.801,388.837,165.576,59.367,160.647
C00887=1014.097,-4.550,388.825,165.578,59.359,160.646
C00888=1014.102,-4.301,388.812,165.580,59.351,160.645
C00889=1014.106,-4.051,388.799,165.583,59.342,160.645
C00890=1014.111,-3.802,388.786,165.585,59.335,160.643
C00891=1014.116,-3.552,388.775,165.586,59.327,160.642
C00892=1014.120,-3.302,388.762,165.589,59.318,160.642
C00893=1014.125,-3.053,388.749,165.591,59.310,160.641
C00894=1014.130,-2.804,388.737,165.594,59.302,160.640
C00895=1014.135,-2.553,388.725,165.596,59.294,160.639
C00896=1014.140,-2.303,388.712,165.598,59.286,160.638
C00897=1014.144,-2.054,388.699,165.600,59.277,160.637
C00898=1014.149,-1.805,388.687,165.602,59.269,160.636
C00899=1014.154,-1.555,388.675,165.605,59.261,160.635
C00900=1014.158,-1.305,388.662,165.607,59.253,160.634
C00901=1014.163,-1.056,388.649,165.609,59.245,160.633
C00902=1014.169,-0.806,388.637,165.612,59.236,160.632
C00903=1014.173,-0.556,388.624,165.613,59.228,160.631
C00904=1014.178,-0.306,388.612,165.616,59.219,160.630
C00905=1014.183,-0.057,388.600,165.618,59.212,160.629
C00906=1014.187,0.192,388.587,165.621,59.203,160.628
C00907=1014.192,0.442,388.574,165.623,59.195,160.627
C00908=1014.197,0.692,388.561,165.625,59.186,160.626
C00909=1014.203,0.941,388.549,165.627,59.178,160.625
C00910=1014.207,1.191,388.537,165.630,59.170,160.624
C00911=1014.211,1.441,388.524,165.632,59.161,160.623
C00912=1014.216,1.690,388.511,165.635,59.153,160.622
C00913=1014.222,1.940,388.499,165.636,59.145,160.621
C00914=1014.226,2.190,388.486,165.639,59.136,160.620
C00915=1014.231,2.439,388.473,165.641,59.128,160.619
C00916=1014.236,2.689,388.460,165.644,59.120,160.618
C00917=1014.241,2.939,388.448,165.645,59.111,160.617
C00918=1014.246,3.189,388.436,165.648,59.103,160.616
C00919=1014.250,3.438,388.423,165.650,59.094,160.615
C00920=1014.256,3.687,388.411,165.652,59.086,160.614
C00921=1014.260,3.937,388.398,165.655,59.077,160.613
C00922=1014.265,4.187,388.385,165.657,59.069,160.612
C00923=1014.270,4.437,388.372,165.660,59.060,160.611
C00924=1014.275,4.686,388.360,165.661,59.052,160.610
C00925=1014.280,4.935,388.347,165.664,59.043,160.609
C00926=1014.285,5.186,388.334,165.666,59.034,160.608
C00927=1014.289,5.435,388.321,165.668,59.026,160.607
C00928=1014.295,5.684,388.309,165.671,59.017,160.606
C00929=1014.299,5.934,388.296,165.673,59.009,160.605
C00930=1014.305,6.184,388.283,165.675,59.000,160.604
C00931=1014.309,6.433,388.270,165.677,58.991,160.602
C00932=1014.314,6.683,388.258,165.679,58.983,160.601
C00933=1014.320,6.933,388.245,165.682,58.974,160.600
C00934=1014.324,7.182,388.232,165.685,58.966,160.600
C00935=1014.329,7.432,388.219,165.686,58.957,160.598
C00936=1014.335,7.682,388.207,165.688,58.948,160.597
C00937=1014.339,7.932,388.195,165.691,58.940,160.596
C00938=1014.344,8.181,388.181,165.693,58.931,160.595
C00939=1014.349,8.430,388.169,165.695,58.922,160.594
C00940=1014.354,8.680,388.156,165.698,58.914,160.593
C00941=1014.359,8.929,388.143,165.701,58.905,160.592
C00942=1014.363,9.179,388.130,165.702,58.896,160.591
C00943=1014.369,9.429,388.118,165.705,58.888,160.590
C00944=1014.374,9.678,388.105,165.707,58.879,160.589
C00945=1014.379,9.958,388.091,165.709,58.869,160.587
C00946=1014.385,10.237,388.077,165.713,58.860,160.586
C00947=1014.390,10.516,388.062,165.714,58.850,160.585
C00948=1014.396,10.795,388.048,165.717,58.840,160.584
C00949=1014.401,11.045,388.035,165.720,58.830,160.583
C00950=1014.406,11.295,388.022,165.722,58.823,160.582
C00951=1014.411,11.545,388.009,165.724,58.814,160.581
C00952=1014.416,11.794,387.997,165.726,58.805,160.580
C00953=1014.421,12.043,387.984,165.729,58.795,160.578
C00954=1014.426,12.294,387.971,165.731,58.786,160.577
C00955=1014.431,12.543,387.958,165.733,58.778,160.576
C00956=1014.436,12.792,387.946,165.735,58.769,160.575
C00957=1014.441,13.043,387.933,165.738,58.760,160.574
C00958=1014.446,13.291,387.919,165.741,58.751,160.573
C00959=1014.451,13.542,387.906,165.742,58.743,160.572
C00960=1014.455,13.791,387.893,165.744,58.734,160.571
C00961=1014.460,14.042,387.879,165.747,58.725,160.570
C00962=1014.465,14.291,387.866,165.749,58.717,160.569
C00963=1014.470,14.540,387.853,165.751,58.708,160.567
C00964=1014.475,14.790,387.840,165.754,58.699,160.566
C00965=1014.479,15.040,387.827,165.757,58.691,160.566
C00966=1014.485,15.289,387.813,165.758,58.682,160.564
C00967=1014.489,15.539,387.801,165.761,58.673,160.563
C00968=1014.495,15.789,387.787,165.763,58.664,160.562
C00969=1014.499,16.038,387.774,165.765,58.655,160.561
C00970=1014.504,16.287,387.761,165.767,58.646,160.560
C00971=1014.509,16.538,387.748,165.770,58.638,160.559
C00972=1014.514,16.786,387.735,165.772,58.629,160.558
C00973=1014.519,17.037,387.721,165.775,58.620,160.557
C00974=1014.524,17.285,387.708,165.776,58.611,160.555
C00975=1014.529,17.536,387.695,165.779,58.602,160.554
C00976=1014.534,17.785,387.682,165.781,58.593,160.553
C00977=1014.539,18.035,387.668,165.784,58.584,160.552
C00978=1014.544,18.284,387.655,165.786,58.575,160.551
C00979=1014.549,18.534,387.642,165.787,58.567,160.550
C00980=1014.554,18.783,387.629,165.790,58.558,160.549
C00981=1014.559,19.033,387.616,165.792,58.549,160.548
C00982=1014.563,19.283,387.601,165.796,58.540,160.547
C00983=1014.568,19.533,387.588,165.798,58.531,160.546
C00984=1014.573,19.782,387.575,165.799,58.523,160.544
C00985=1014.578,20.032,387.562,165.802,58.514,160.543
C00986=1014.583,20.281,387.548,165.804,58.505,160.542
C00987=1014.588,20.531,387.534,165.807,58.496,160.541
C00988=1014.593,20.780,387.521,165.808,58.487,160.540
C00989=1014.598,21.030,387.508,165.811,58.478,160.539
C00990=1014.603,21.279,387.494,165.813,58.469,160.538
C00991=1014.608,21.529,387.481,165.816,58.460,160.537
C00992=1014.612,21.779,387.467,165.818,58.451,160.535
C00993=1014.617,22.028,387.453,165.820,58.443,160.534
C00994=1014.622,22.278,387.440,165.822,58.434,160.533
C00995=1014.628,22.527,387.427,165.825,58.425,160.532
C00996=1014.632,22.777,387.414,165.827,58.416,160.531
C00997=1014.637,23.027,387.399,165.830,58.407,160.530
C00998=1014.641,23.276,387.386,165.832,58.398,160.529
C00999=1014.647,23.526,387.373,165.835,58.389,160.528
C01000=1014.651,23.775,387.360,165.836,58.380,160.526
C01001=1014.657,24.025,387.346,165.838,58.370,160.525
C01002=1014.662,24.275,387.332,165.841,58.361,160.524
C01003=1014.666,24.524,387.319,165.843,58.352,160.523
C01004=1014.672,24.774,387.305,165.846,58.343,160.522
C01005=1014.676,25.023,387.292,165.848,58.334,160.521
C01006=1014.682,25.273,387.278,165.851,58.325,160.520
C01007=1014.686,25.522,387.264,165.853,58.316,160.518
C01008=1014.691,25.772,387.251,165.854,58.307,160.517
C01009=1014.697,26.053,387.235,165.857,58.297,160.516
C01010=1014.703,26.334,387.220,165.860,58.287,160.514
C01011=1014.708,26.615,387.204,165.863,58.277,160.513
C01012=1014.713,26.895,387.190,165.865,58.267,160.512
C01013=1014.718,27.145,387.176,165.867,58.257,160.510
C01014=1014.724,27.394,387.162,165.869,58.248,160.509
C01015=1014.728,27.644,387.148,165.872,58.239,160.508
C01016=1014.733,27.894,387.135,165.874,58.230,160.507
C01017=1014.738,28.144,387.120,165.877,58.221,160.506
C01018=1014.743,28.393,387.107,165.880,58.212,160.505
C01019=1014.748,28.642,387.092,165.881,58.204,160.504
C01020=1014.752,28.891,387.079,165.884,58.195,160.503
C01021=1014.757,29.142,387.065,165.886,58.185,160.501
C01022=1014.762,29.391,387.051,165.888,58.176,160.500
C01023=1014.767,29.640,387.038,165.891,58.167,160.499
C01024=1014.772,29.890,387.023,165.893,58.158,160.498
C01025=1014.777,30.140,387.009,165.896,58.149,160.497
C01026=1014.782,30.389,386.995,165.898,58.140,160.496
C01027=1014.787,30.638,386.981,165.899,58.131,160.494
C01028=1014.791,30.889,386.967,165.902,58.122,160.493
C01029=1014.796,31.138,386.954,165.904,58.113,160.492
C01030=1014.801,31.388,386.940,165.906,58.103,160.491
C01031=1014.807,31.637,386.926,165.909,58.095,160.490
C01032=1014.811,31.887,386.912,165.911,58.086,160.489
C01033=1014.816,32.136,386.898,165.914,58.077,160.488
C01034=1014.822,32.386,386.884,165.916,58.067,160.486
C01035=1014.826,32.635,386.870,165.919,58.058,160.485
C01036=1014.831,32.884,386.856,165.921,58.049,160.484
C01037=1014.836,33.135,386.842,165.923,58.039,160.483
C01038=1014.841,33.384,386.829,165.926,58.030,160.482
C01039=1014.845,33.634,386.814,165.928,58.021,160.481
C01040=1014.851,33.883,386.800,165.930,58.012,160.479
C01041=1014.855,34.133,386.786,165.933,58.003,160.478
C01042=1014.860,34.382,386.772,165.935,57.993,160.477
C01043=1014.865,34.632,386.758,165.938,57.984,160.476
C01044=1014.871,34.881,386.744,165.940,57.975,160.475
C01045=1014.875,35.131,386.730,165.942,57.966,160.473
C01046=1014.880,35.380,386.716,165.945,57.957,160.472
C01047=1014.886,35.630,386.702,165.947,57.947,160.471
C01048=1014.890,35.880,386.688,165.949,57.938,160.470
C01049=1014.895,36.129,386.674,165.951,57.928,160.468
C01050=1014.900,36.378,386.660,165.954,57.919,160.467
C01051=1014.905,36.628,386.645,165.957,57.911,160.466
C01052=1014.910,36.878,386.631,165.958,57.901,160.465
C01053=1014.915,37.128,386.617,165.960,57.892,160.464
C01054=1014.919,37.377,386.603,165.963,57.883,160.463
C01055=1014.924,37.626,386.588,165.965,57.874,160.461
C01056=1014.930,37.876,386.574,165.967,57.865,160.460
C01057=1014.934,38.126,386.559,165.970,57.856,160.459
C01058=1014.939,38.375,386.545,165.972,57.846,160.458
C01059=1014.944,38.624,386.531,165.975,57.837,160.457
C01060=1014.949,38.874,386.517,165.977,57.828,160.455
C01061=1014.954,39.124,386.502,165.979,57.819,160.454
C01062=1014.958,39.374,386.487,165.981,57.809,160.453
C01063=1014.963,39.622,386.474,165.984,57.800,160.452
C01064=1014.968,39.872,386.459,165.987,57.791,160.451
C01065=1014.973,40.122,386.445,165.989,57.782,160.449
C01066=1014.978,40.372,386.431,165.991,57.773,160.448
C01067=1014.983,40.621,386.416,165.993,57.763,160.447
C01068=1014.988,40.870,386.402,165.996,57.754,160.446
C01069=1014.992,41.120,386.387,165.998,57.745,160.445
C01070=1014.998,41.370,386.374,166.001,57.736,160.444
C01071=1015.003,41.619,386.358,166.003,57.726,160.442
C01072=1015.007,41.869,386.344,166.005,57.717,160.441
C01073=1015.013,42.150,386.328,166.008,57.706,160.440
C01074=1015.018,42.431,386.311,166.010,57.697,160.438
C01075=1015.024,42.711,386.295,166.013,57.686,160.437
C01076=1015.029,42.993,386.278,166.016,57.676,160.436
C01077=1015.034,43.242,386.263,166.018,57.666,160.434
C01078=1015.038,43.491,386.249,166.020,57.657,160.433
C01079=1015.043,43.741,386.234,166.023,57.648,160.432
C01080=1015.048,43.991,386.220,166.025,57.639,160.431
C01081=1015.053,44.240,386.204,166.028,57.630,160.430
C01082=1015.058,44.490,386.190,166.029,57.621,160.428
C01083=1015.063,44.739,386.175,166.032,57.612,160.427
C01084=1015.067,44.989,386.160,166.034,57.603,160.426
C01085=1015.072,45.238,386.146,166.036,57.593,160.425
C01086=1015.077,45.487,386.131,166.039,57.584,160.424
C01087=1015.081,45.737,386.117,166.041,57.575,160.422
C01088=1015.086,45.987,386.101,166.044,57.566,160.421
C01089=1015.091,46.236,386.087,166.046,57.556,160.420
C01090=1015.096,46.486,386.072,166.049,57.547,160.419
C01091=1015.101,46.736,386.057,166.051,57.538,160.418
C01092=1015.106,46.985,386.042,166.053,57.529,160.417
C01093=1015.111,47.235,386.028,166.055,57.519,160.415
C01094=1015.116,47.484,386.012,166.058,57.510,160.414
C01095=1015.120,47.733,385.998,166.060,57.501,160.413
C01096=1015.125,47.982,385.983,166.062,57.491,160.411
C01097=1015.130,48.232,385.969,166.065,57.482,160.410
C01098=1015.135,48.482,385.954,166.067,57.473,160.409
C01099=1015.139,48.731,385.939,166.070,57.464,160.408
C01100=1015.145,48.981,385.924,166.072,57.454,160.407
C01101=1015.150,49.230,385.909,166.075,57.445,160.406
C01102=1015.154,49.480,385.894,166.077,57.436,160.404
C01103=1015.159,49.729,385.879,166.079,57.426,160.403
C01104=1015.164,49.979,385.865,166.082,57.417,160.402
C01105=1015.169,50.228,385.850,166.084,57.408,160.401
C01106=1015.174,50.478,385.835,166.086,57.398,160.399
C01107=1015.179,50.727,385.820,166.089,57.389,160.398
C01108=1015.184,50.977,385.805,166.091,57.380,160.397
C01109=1015.189,51.227,385.790,166.093,57.370,160.396
C01110=1015.194,51.476,385.775,166.097,57.361,160.395
C01111=1015.198,51.726,385.761,166.099,57.351,160.393
C01112=1015.204,51.975,385.745,166.101,57.342,160.392
C01113=1015.209,52.224,385.730,166.103,57.332,160.391
C01114=1015.213,52.474,385.716,166.106,57.323,160.390
C01115=1015.218,52.723,385.701,166.108,57.314,160.388
C01116=1015.223,52.973,385.686,166.110,57.304,160.387
C01117=1015.228,53.223,385.671,166.112,57.295,160.386
C01118=1015.232,53.472,385.655,166.115,57.286,160.385
C01119=1015.237,53.722,385.641,166.117,57.276,160.383
C01120=1015.242,53.971,385.626,166.120,57.267,160.382
C01121=1015.247,54.221,385.610,166.123,57.257,160.381
C01122=1015.252,54.470,385.596,166.125,57.247,160.379
C01123=1015.257,54.720,385.581,166.128,57.238,160.378
C01124=1015.262,54.969,385.566,166.130,57.229,160.377
C01125=1015.267,55.219,385.551,166.132,57.219,160.376
C01126=1015.272,55.468,385.536,166.134,57.210,160.374
C01127=1015.277,55.717,385.521,166.136,57.200,160.373
C01128=1015.282,55.967,385.506,166.140,57.190,160.372
C01129=1015.287,56.217,385.491,166.142,57.181,160.371
C01130=1015.292,56.466,385.476,166.145,57.172,160.370
C01131=1015.296,56.716,385.462,166.147,57.162,160.368
C01132=1015.302,56.965,385.446,166.149,57.152,160.367
C01133=1015.307,57.214,385.431,166.151,57.143,160.366
C01134=1015.312,57.464,385.416,166.155,57.133,160.365
C01135=1015.316,57.713,385.402,166.157,57.123,160.363
C01136=1015.321,57.963,385.386,166.159,57.114,160.362
C01137=1015.327,58.244,385.369,166.162,57.103,160.360
C01138=1015.333,58.525,385.353,166.164,57.092,160.359
C01139=1015.338,58.806,385.335,166.167,57.082,160.358
C01140=1015.344,59.086,385.319,166.170,57.071,160.356
C01141=1015.349,59.336,385.304,166.173,57.061,160.355
C01142=1015.354,59.586,385.288,166.175,57.052,160.354
C01143=1015.359,59.835,385.273,166.177,57.042,160.352
C01144=1015.364,60.085,385.258,166.180,57.032,160.351
C01145=1015.369,60.334,385.243,166.183,57.022,160.350
C01146=1015.374,60.584,385.228,166.185,57.013,160.349
C01147=1015.379,60.833,385.213,166.187,57.003,160.347
C01148=1015.384,61.082,385.198,166.190,56.994,160.346
C01149=1015.389,61.332,385.183,166.193,56.984,160.345
C01150=1015.394,61.581,385.168,166.195,56.974,160.344
C01151=1015.399,61.831,385.152,166.197,56.965,160.342
C01152=1015.404,62.080,385.137,166.199,56.955,160.341
C01153=1015.410,62.330,385.122,166.202,56.945,160.340
C01154=1015.414,62.580,385.108,166.205,56.935,160.338
C01155=1015.419,62.829,385.092,166.207,56.926,160.337
C01156=1015.424,63.078,385.077,166.209,56.916,160.336
C01157=1015.429,63.328,385.061,166.212,56.907,160.335
C01158=1015.434,63.578,385.046,166.214,56.898,160.333
C01159=1015.439,63.827,385.030,166.218,56.888,160.332
C01160=1015.444,64.077,385.015,166.220,56.878,160.331
C01161=1015.449,64.326,385.000,166.222,56.869,160.329
C01162=1015.453,64.575,384.983,166.224,56.859,160.328
C01163=1015.459,64.825,384.968,166.227,56.850,160.327
C01164=1015.464,65.074,384.953,166.229,56.840,160.326
C01165=1015.468,65.324,384.937,166.232,56.830,160.324
C01166=1015.473,65.573,384.922,166.234,56.821,160.323
C01167=1015.478,65.822,384.906,166.237,56.811,160.322
C01168=1015.483,66.072,384.890,166.239,56.802,160.321
C01169=1015.489,66.369,384.872,166.242,56.790,160.319
C01170=1015.494,66.665,384.853,166.245,56.779,160.318
C01171=1015.501,66.962,384.835,166.248,56.768,160.316
C01172=1015.507,67.258,384.816,166.251,56.756,160.314
C01173=1015.511,67.508,384.801,166.253,56.747,160.313
C01174=1015.516,67.757,384.786,166.256,56.737,160.312
C01175=1015.521,68.007,384.769,166.259,56.727,160.311
C01176=1015.526,68.257,384.754,166.261,56.718,160.309
C01177=1015.530,68.506,384.738,166.263,56.708,160.308
C01178=1015.536,68.755,384.723,166.266,56.700,160.307
C01179=1015.540,69.004,384.707,166.268,56.690,160.306
C01180=1015.546,69.254,384.691,166.272,56.680,160.305
C01181=1015.550,69.504,384.675,166.274,56.671,160.303
C01182=1015.555,69.753,384.660,166.276,56.661,160.302
C01183=1015.560,70.002,384.644,166.279,56.652,160.301
C01184=1015.564,70.252,384.628,166.281,56.642,160.299
C01185=1015.569,70.502,384.613,166.283,56.633,160.298
C01186=1015.574,70.751,384.596,166.287,56.623,160.297
C01187=1015.579,71.000,384.581,166.289,56.613,160.296
C01188=1015.584,71.250,384.565,166.291,56.604,160.294
C01189=1015.589,71.499,384.548,166.294,56.595,160.293
C01190=1015.594,71.748,384.533,166.296,56.585,160.292
C01191=1015.599,71.999,384.517,166.298,56.576,160.291
C01192=1015.604,72.247,384.501,166.302,56.566,160.289
C01193=1015.608,72.497,384.485,166.303,56.555,160.288
C01194=1015.613,72.746,384.470,166.306,56.546,160.287
C01195=1015.619,72.996,384.453,166.308,56.537,160.285
C01196=1015.623,73.245,384.437,166.311,56.527,160.284
C01197=1015.627,73.487,384.422,166.313,56.518,160.283
C01198=1015.632,73.729,384.406,166.316,56.509,160.282
C01199=1015.637,73.970,384.392,166.318,56.499,160.280
C01200=1015.642,74.212,384.377,166.320,56.490,160.279
C01201=1015.647,74.453,384.361,166.323,56.481,160.278
C01202=1015.652,74.695,384.346,166.325,56.471,160.277
C01203=1015.656,74.936,384.330,166.328,56.462,160.276
C01204=1015.661,75.178,384.314,166.330,56.453,160.274
C01205=1015.666,75.428,384.299,166.334,56.443,160.273
C01206=1015.672,75.677,384.282,166.336,56.433,160.272
C01207=1015.676,75.927,384.267,166.338,56.423,160.270
C01208=1015.680,76.176,384.251,166.340,56.414,160.269
C01209=1015.685,76.426,384.234,166.343,56.405,160.268
C01210=1015.690,76.675,384.219,166.346,56.395,160.267
C01211=1015.695,76.924,384.202,166.349,56.385,160.265
C01212=1015.700,77.175,384.186,166.351,56.376,160.264
C01213=1015.705,77.424,384.170,166.353,56.366,160.263
C01214=1015.709,77.672,384.153,166.356,56.357,160.262
C01215=1015.714,77.923,384.137,166.359,56.347,160.260
C01216=1015.719,78.171,384.121,166.362,56.338,160.259
C01217=1015.724,78.421,384.105,166.364,56.328,160.258
C01218=1015.729,78.671,384.089,166.366,56.319,160.257
C01219=1015.734,78.920,384.072,166.369,56.309,160.255
C01220=1015.738,79.169,384.056,166.371,56.300,160.254
C01221=1015.743,79.419,384.040,166.375,56.290,160.253
C01222=1015.747,79.668,384.024,166.377,56.281,160.252
C01223=1015.753,79.918,384.007,166.380,56.271,160.250
C01224=1015.757,80.167,383.990,166.382,56.262,160.249
C01225=1015.762,80.416,383.975,166.384,56.252,160.248
C01226=1015.768,80.666,383.958,166.386,56.242,160.246
C01227=1015.772,80.915,383.942,166.390,56.232,160.245
C01228=1015.777,81.165,383.926,166.392,56.223,160.244
C01229=1015.782,81.414,383.909,166.395,56.214,160.243
C01230=1015.786,81.663,383.893,166.397,56.204,160.241
C01231=1015.791,81.913,383.877,166.399,56.195,160.240
C01232=1015.796,82.162,383.860,166.403,56.185,160.239
C01233=1015.801,82.412,383.843,166.405,56.175,160.237
C01234=1015.806,82.661,383.828,166.407,56.165,160.236
C01235=1015.811,82.911,383.811,166.410,56.156,160.235
C01236=1015.816,83.160,383.795,166.413,56.146,160.234
C01237=1015.820,83.409,383.779,166.416,56.137,160.232
C01238=1015.825,83.659,383.762,166.418,56.127,160.231
C01239=1015.830,83.908,383.746,166.420,56.117,160.230
C01240=1015.835,84.158,383.729,166.423,56.107,160.229
C01241=1015.840,84.407,383.713,166.426,56.098,160.227
C01242=1015.845,84.657,383.696,166.428,56.089,160.226
C01243=1015.849,84.906,383.680,166.431,56.079,160.225
C01244=1015.855,85.155,383.663,166.434,56.069,160.223
C01245=1015.860,85.405,383.648,166.436,56.059,160.222
C01246=1015.865,85.655,383.631,166.439,56.050,160.221
C01247=1015.869,85.903,383.614,166.442,56.040,160.220
C01248=1015.875,86.153,383.598,166.444,56.030,160.218
C01249=1015.879,86.403,383.582,166.447,56.021,160.217
C01250=1015.884,86.652,383.565,166.449,56.011,160.216
C01251=1015.889,86.901,383.548,166.453,56.001,160.215
C01252=1015.894,87.151,383.532,166.454,55.991,160.213
C01253=1015.899,87.400,383.515,166.457,55.982,160.212
C01254=1015.904,87.650,383.500,166.461,55.972,160.211
C01255=1015.909,87.899,383.483,166.462,55.962,160.209
C01256=1015.914,88.149,383.466,166.465,55.953,160.208
C01257=1015.919,88.398,383.450,166.468,55.943,160.207
C01258=1015.924,88.647,383.433,166.470,55.933,160.205
C01259=1015.928,88.896,383.416,166.473,55.923,160.204
C01260=1015.933,89.146,383.400,166.475,55.914,160.203
C01261=1015.937,89.396,383.383,166.479,55.904,160.202
C01262=1015.942,89.645,383.366,166.481,55.895,160.200
C01263=1015.947,89.894,383.350,166.484,55.886,160.199
C01264=1015.952,90.144,383.333,166.486,55.876,160.198
C01265=1015.958,90.425,383.314,166.489,55.865,160.196
C01266=1015.963,90.706,383.295,166.492,55.854,160.195
C01267=1015.969,90.987,383.276,166.496,55.844,160.194
C01268=1015.974,91.268,383.257,166.499,55.832,160.192
C01269=1015.978,91.517,383.240,166.501,55.823,160.191
C01270=1015.983,91.767,383.223,166.504,55.814,160.190
C01271=1015.988,92.016,383.206,166.506,55.804,160.188
C01272=1015.993,92.265,383.190,166.509,55.794,160.187
C01273=1015.998,92.515,383.173,166.512,55.784,160.186
C01274=1016.002,92.764,383.156,166.514,55.775,160.184
C01275=1016.007,93.014,383.139,166.517,55.766,160.183
C01276=1016.012,93.262,383.122,166.520,55.756,160.182
C01277=1016.018,93.512,383.105,166.522,55.746,160.181
C01278=1016.021,93.761,383.088,166.525,55.737,160.179
C01279=1016.027,94.011,383.071,166.528,55.727,160.178
C01280=1016.032,94.261,383.054,166.531,55.718,160.177
C01281=1016.036,94.510,383.037,166.533,55.707,160.176
C01282=1016.042,94.759,383.021,166.535,55.698,160.174
C01283=1016.046,95.008,383.004,166.539,55.688,160.173
C01284=1016.051,95.258,382.987,166.541,55.678,160.172
C01285=1016.056,95.507,382.969,166.544,55.669,160.170
C01286=1016.061,95.756,382.953,166.547,55.659,160.169
C01287=1016.065,96.006,382.935,166.550,55.650,160.168
C01288=1016.071,96.256,382.918,166.552,55.640,160.167
C01289=1016.075,96.505,382.902,166.554,55.631,160.165
C01290=1016.080,96.754,382.885,166.558,55.621,160.164
C01291=1016.086,97.004,382.868,166.560,55.611,160.163
C01292=1016.090,97.253,382.850,166.563,55.601,160.161
C01293=1016.095,97.502,382.833,166.566,55.592,160.160
C01294=1016.100,97.751,382.817,166.568,55.582,160.159
C01295=1016.105,98.001,382.800,166.571,55.572,160.158
C01296=1016.109,98.251,382.783,166.574,55.563,160.157
C01297=1016.114,98.499,382.765,166.577,55.553,160.155
C01298=1016.119,98.749,382.749,166.579,55.543,160.154
C01299=1016.125,98.999,382.732,166.582,55.533,160.152
C01300=1016.129,99.249,382.714,166.585,55.524,160.151
C01301=1016.134,99.497,382.697,166.587,55.514,160.150
C01302=1016.139,99.747,382.680,166.590,55.505,160.149
C01303=1016.143,99.996,382.662,166.594,55.495,160.148
C01304=1016.148,100.245,382.645,166.596,55.485,160.146
C01305=1016.152,100.495,382.628,166.598,55.476,160.145
C01306=1016.158,100.744,382.610,166.601,55.467,160.144
C01307=1016.162,100.993,382.593,166.604,55.457,160.143
C01308=1016.167,101.243,382.575,166.607,55.448,160.141
C01309=1016.172,101.492,382.558,166.609,55.438,160.140
C01310=1016.176,101.741,382.541,166.612,55.428,160.139
C01311=1016.181,101.991,382.523,166.615,55.419,160.138
C01312=1016.186,102.240,382.506,166.618,55.409,160.136
C01313=1016.191,102.490,382.488,166.620,55.399,160.135
C01314=1016.196,102.739,382.472,166.624,55.390,160.134
C01315=1016.201,102.988,382.454,166.626,55.380,160.133
C01316=1016.206,103.238,382.437,166.629,55.370,160.131
C01317=1016.210,103.486,382.419,166.631,55.361,160.130
C01318=1016.215,103.736,382.402,166.635,55.351,160.129
C01319=1016.220,103.986,382.385,166.637,55.342,160.127
C01320=1016.225,104.235,382.367,166.640,55.332,160.126
C01321=1016.229,104.484,382.350,166.643,55.322,160.125
C01322=1016.234,104.734,382.332,166.646,55.313,160.124
C01323=1016.239,104.983,382.315,166.648,55.303,160.122
C01324=1016.244,105.233,382.297,166.652,55.293,160.121
C01325=1016.248,105.482,382.280,166.654,55.284,160.120
C01326=1016.253,105.731,382.262,166.656,55.274,160.118
C01327=1016.259,105.980,382.245,166.660,55.265,160.117
C01328=1016.263,106.230,382.227,166.663,55.255,160.116
C01329=1016.268,106.511,382.208,166.665,55.244,160.114
C01330=1016.274,106.792,382.188,166.668,55.233,160.113
C01331=1016.280,107.074,382.168,166.672,55.222,160.112
C01332=1016.285,107.355,382.148,166.675,55.211,160.110
C01333=1016.290,107.604,382.131,166.678,55.202,160.109
C01334=1016.294,107.854,382.114,166.681,55.192,160.108
C01335=1016.300,108.103,382.096,166.683,55.182,160.106
C01336=1016.305,108.352,382.078,166.686,55.173,160.105
C01337=1016.310,108.602,382.061,166.689,55.163,160.104
C01338=1016.314,108.850,382.043,166.692,55.153,160.103
C01339=1016.319,109.100,382.027,166.696,55.144,160.102
C01340=1016.324,109.349,382.008,166.698,55.134,160.100
C01341=1016.329,109.599,381.990,166.701,55.125,160.099
C01342=1016.333,109.849,381.973,166.704,55.115,160.098
C01343=1016.339,110.098,381.955,166.706,55.105,160.096
C01344=1016.343,110.346,381.937,166.709,55.096,160.095
C01345=1016.348,110.596,381.919,166.713,55.086,160.094
C01346=1016.353,110.845,381.902,166.715,55.076,160.092
C01347=1016.358,111.095,381.884,166.718,55.067,160.091
C01348=1016.363,111.344,381.866,166.721,55.057,160.090
C01349=1016.367,111.594,381.849,166.724,55.047,160.089
C01350=1016.373,111.843,381.831,166.726,55.038,160.087
C01351=1016.377,112.092,381.813,166.730,55.028,160.086
C01352=1016.382,112.341,381.795,166.732,55.018,160.085
C01353=1016.386,112.590,381.777,166.735,55.009,160.084
C01354=1016.391,112.840,381.759,166.738,55.000,160.082
C01355=1016.396,113.089,381.741,166.740,54.991,160.081
C01356=1016.401,113.339,381.722,166.744,54.981,160.080
C01357=1016.406,113.588,381.704,166.746,54.971,160.079
C01358=1016.409,113.837,381.687,166.749,54.962,160.078
C01359=1016.414,114.087,381.669,166.752,54.953,160.076
C01360=1016.419,114.336,381.651,166.756,54.943,160.075
C01361=1016.424,114.585,381.633,166.758,54.934,160.074
C01362=1016.429,114.835,381.615,166.760,54.924,160.073
C01363=1016.433,115.084,381.596,166.764,54.914,160.071
C01364=1016.438,115.333,381.578,166.767,54.905,160.070
C01365=1016.443,115.583,381.560,166.770,54.896,160.069
C01366=1016.448,115.832,381.542,166.772,54.886,160.068
C01367=1016.452,116.081,381.524,166.776,54.876,160.067
C01368=1016.456,116.330,381.505,166.778,54.867,160.065
C01369=1016.461,116.580,381.487,166.781,54.858,160.064
C01370=1016.465,116.829,381.469,166.784,54.848,160.063
C01371=1016.470,117.078,381.451,166.787,54.838,160.062
C01372=1016.475,117.328,381.433,166.790,54.829,160.060
C01373=1016.480,117.577,381.415,166.793,54.820,160.059
C01374=1016.485,117.826,381.396,166.796,54.810,160.058
C01375=1016.489,118.076,381.378,166.799,54.801,160.057
C01376=1016.494,118.324,381.359,166.801,54.791,160.055
C01377=1016.499,118.574,381.341,166.805,54.781,160.054
C01378=1016.504,118.823,381.323,166.808,54.772,160.053
C01379=1016.509,119.073,381.305,166.810,54.763,160.052
C01380=1016.514,119.322,381.287,166.814,54.752,160.050
C01381=1016.518,119.571,381.269,166.816,54.743,160.049
C01382=1016.523,119.821,381.250,166.819,54.734,160.048
C01383=1016.528,120.070,381.232,166.822,54.724,160.047
C01384=1016.533,120.319,381.214,166.825,54.715,160.045
C01385=1016.537,120.569,381.196,166.829,54.705,160.044
C01386=1016.542,120.818,381.178,166.831,54.695,160.043
C01387=1016.547,121.067,381.159,166.834,54.686,160.042
C01388=1016.552,121.316,381.141,166.838,54.676,160.041
C01389=1016.557,121.565,381.123,166.840,54.666,160.039
C01390=1016.562,121.815,381.104,166.843,54.657,160.038
C01391=1016.566,122.064,381.086,166.847,54.648,160.037
C01392=1016.571,122.313,381.068,166.849,54.638,160.035
C01393=1016.577,122.595,381.047,166.852,54.628,160.034
C01394=1016.582,122.876,381.027,166.856,54.616,160.033
C01395=1016.588,123.157,381.006,166.859,54.605,160.031
C01396=1016.592,123.439,380.985,166.863,54.595,160.030
C01397=1016.597,123.688,380.967,166.866,54.585,160.029
C01398=1016.602,123.937,380.949,166.869,54.575,160.027
C01399=1016.607,124.186,380.930,166.872,54.566,160.026
C01400=1016.612,124.435,380.912,166.875,54.556,160.025
C01401=1016.617,124.685,380.893,166.879,54.547,160.024
C01402=1016.621,124.934,380.875,166.881,54.537,160.022
C01403=1016.627,125.184,380.857,166.884,54.528,160.021
C01404=1016.632,125.433,380.838,166.888,54.518,160.020
C01405=1016.637,125.682,380.820,166.890,54.508,160.019
C01406=1016.641,125.932,380.802,166.894,54.499,160.018
C01407=1016.646,126.181,380.783,166.896,54.489,160.016
C01408=1016.651,126.430,380.764,166.900,54.479,160.015
C01409=1016.656,126.679,380.746,166.902,54.469,160.014
C01410=1016.661,126.928,380.728,166.906,54.460,160.013
C01411=1016.666,127.178,380.710,166.909,54.451,160.011
C01412=1016.671,127.426,380.691,166.912,54.440,160.010
C01413=1016.676,127.676,380.673,166.915,54.431,160.009
C01414=1016.681,127.926,380.654,166.918,54.421,160.007
C01415=1016.686,128.175,380.636,166.921,54.412,160.006
C01416=1016.691,128.424,380.617,166.924,54.402,160.005
C01417=1016.696,128.673,380.599,166.928,54.393,160.004
C01418=1016.701,128.922,380.580,166.930,54.383,160.002
C01419=1016.705,129.172,380.562,166.934,54.373,160.001
C01420=1016.709,129.421,380.543,166.936,54.363,160.000
C01421=1016.715,129.670,380.524,166.940,54.354,159.999
C01422=1016.720,129.920,380.506,166.943,54.345,159.998
C01423=1016.724,130.169,380.487,166.946,54.334,159.996
C01424=1016.729,130.418,380.468,166.949,54.325,159.995
C01425=1016.734,130.667,380.450,166.952,54.316,159.994
C01426=1016.739,130.917,380.430,166.955,54.306,159.993
C01427=1016.744,131.166,380.412,166.958,54.297,159.991
C01428=1016.748,131.416,380.393,166.961,54.288,159.990
C01429=1016.753,131.664,380.374,166.965,54.278,159.989
C01430=1016.758,131.914,380.356,166.968,54.268,159.988
C01431=1016.762,132.163,380.336,166.971,54.259,159.987
C01432=1016.768,132.412,380.317,166.974,54.250,159.986
C01433=1016.772,132.662,380.298,166.977,54.240,159.984
C01434=1016.777,132.911,380.279,166.981,54.231,159.983
C01435=1016.782,133.160,380.261,166.983,54.221,159.982
C01436=1016.786,133.409,380.242,166.987,54.211,159.981
C01437=1016.792,133.658,380.223,166.990,54.202,159.979
C01438=1016.796,133.908,380.204,166.994,54.193,159.978
C01439=1016.801,134.157,380.185,166.996,54.183,159.977
C01440=1016.806,134.406,380.167,166.999,54.174,159.976
C01441=1016.810,134.655,380.147,167.002,54.164,159.974
C01442=1016.816,134.905,380.128,167.005,54.155,159.973
C01443=1016.820,135.154,380.109,167.009,54.145,159.972
C01444=1016.825,135.403,380.090,167.012,54.135,159.971
C01445=1016.829,135.652,380.071,167.016,54.126,159.970
C01446=1016.835,135.902,380.052,167.019,54.117,159.969
C01447=1016.839,136.151,380.033,167.021,54.107,159.967
C01448=1016.844,136.400,380.014,167.025,54.097,159.966
C01449=1016.848,136.649,379.995,167.028,54.088,159.965
C01450=1016.854,136.899,379.976,167.031,54.078,159.964
C01451=1016.858,137.148,379.957,167.034,54.069,159.962
C01452=1016.863,137.397,379.938,167.038,54.060,159.961
C01453=1016.868,137.646,379.918,167.041,54.050,159.960
C01454=1016.873,137.896,379.900,167.045,54.040,159.959
C01455=1016.877,138.145,379.880,167.047,54.031,159.958
C01456=1016.882,138.394,379.861,167.050,54.022,159.956
C01457=1016.888,138.675,379.839,167.054,54.011,159.955
C01458=1016.893,138.956,379.817,167.058,54.001,159.954
C01459=1016.898,139.238,379.796,167.061,53.990,159.952
C01460=1016.903,139.519,379.774,167.065,53.979,159.951
C01461=1016.909,139.768,379.755,167.068,53.970,159.950
C01462=1016.913,140.017,379.735,167.072,53.960,159.949
C01463=1016.918,140.267,379.715,167.075,53.951,159.947
C01464=1016.923,140.516,379.696,167.078,53.942,159.946
C01465=1016.927,140.765,379.677,167.081,53.932,159.945
C01466=1016.932,141.014,379.657,167.084,53.923,159.944
C01467=1016.937,141.264,379.639,167.088,53.913,159.943
C01468=1016.941,141.513,379.620,167.091,53.904,159.942
C01469=1016.946,141.762,379.600,167.095,53.894,159.940
C01470=1016.951,142.011,379.581,167.098,53.885,159.939
C01471=1016.956,142.260,379.561,167.102,53.876,159.938
C01472=1016.961,142.510,379.541,167.104,53.866,159.937
C01473=1016.966,142.759,379.523,167.108,53.857,159.936
C01474=1016.970,143.008,379.503,167.111,53.848,159.934
C01475=1016.975,143.257,379.483,167.115,53.837,159.933
C01476=1016.980,143.506,379.464,167.118,53.828,159.932
C01477=1016.985,143.756,379.445,167.120,53.819,159.931
C01478=1016.989,144.005,379.425,167.124,53.809,159.930
C01479=1016.995,144.254,379.406,167.127,53.800,159.928
C01480=1017.000,144.503,379.386,167.131,53.791,159.927
C01481=1017.004,144.753,379.367,167.133,53.781,159.926
C01482=1017.010,145.001,379.347,167.138,53.772,159.925
C01483=1017.014,145.250,379.328,167.140,53.763,159.924
C01484=1017.019,145.499,379.308,167.145,53.753,159.923
C01485=1017.023,145.749,379.288,167.147,53.744,159.921
C01486=1017.028,145.998,379.269,167.151,53.734,159.920
C01487=1017.034,146.248,379.249,167.154,53.725,159.919
C01488=1017.038,146.497,379.230,167.158,53.716,159.918
C01489=1017.042,146.746,379.211,167.161,53.706,159.917
C01490=1017.047,146.995,379.190,167.165,53.697,159.915
C01491=1017.052,147.244,379.171,167.168,53.688,159.914
C01492=1017.057,147.494,379.151,167.172,53.678,159.913
C01493=1017.061,147.743,379.131,167.174,53.668,159.912
C01494=1017.066,147.992,379.111,167.178,53.659,159.911
C01495=1017.071,148.241,379.091,167.181,53.650,159.910
C01496=1017.075,148.490,379.072,167.185,53.641,159.909
C01497=1017.081,148.739,379.052,167.188,53.631,159.907
C01498=1017.085,148.988,379.032,167.192,53.622,159.906
C01499=1017.090,149.237,379.012,167.195,53.613,159.905
C01500=1017.095,149.487,378.993,167.198,53.604,159.904
C01501=1017.100,149.736,378.972,167.202,53.594,159.903
C01502=1017.104,149.985,378.953,167.204,53.585,159.901
C01503=1017.109,150.234,378.933,167.209,53.575,159.900
C01504=1017.114,150.483,378.913,167.212,53.566,159.899
C01505=1017.119,150.733,378.893,167.216,53.557,159.898
C01506=1017.123,150.982,378.874,167.218,53.547,159.897
C01507=1017.128,151.231,378.853,167.222,53.538,159.896
C01508=1017.133,151.480,378.834,167.225,53.529,159.894
C01509=1017.138,151.730,378.814,167.229,53.519,159.893
C01510=1017.142,151.978,378.794,167.232,53.510,159.892
C01511=1017.147,152.228,378.774,167.236,53.500,159.891
C01512=1017.152,152.476,378.754,167.240,53.491,159.890
C01513=1017.157,152.726,378.734,167.243,53.482,159.889
C01514=1017.161,152.975,378.714,167.247,53.472,159.887
C01515=1017.167,153.224,378.694,167.250,53.463,159.886
C01516=1017.172,153.474,378.674,167.254,53.454,159.885
C01517=1017.176,153.722,378.654,167.257,53.445,159.884
C01518=1017.181,153.972,378.634,167.261,53.435,159.883
C01519=1017.186,154.220,378.614,167.264,53.426,159.882
C01520=1017.190,154.470,378.593,167.268,53.416,159.881
C01521=1017.195,154.751,378.571,167.271,53.406,159.879
C01522=1017.201,155.032,378.548,167.276,53.396,159.878
C01523=1017.206,155.314,378.525,167.279,53.385,159.877
C01524=1017.212,155.595,378.502,167.283,53.375,159.875
C01525=1017.217,155.844,378.482,167.287,53.366,159.874
C01526=1017.222,156.093,378.462,167.290,53.356,159.873
C01527=1017.226,156.342,378.442,167.293,53.347,159.872
C01528=1017.231,156.591,378.422,167.298,53.337,159.871
C01529=1017.236,156.841,378.402,167.301,53.328,159.870
C01530=1017.240,157.089,378.381,167.305,53.319,159.869
C01531=1017.245,157.339,378.361,167.307,53.309,159.867
C01532=1017.250,157.588,378.341,167.312,53.300,159.866
C01533=1017.255,157.837,378.320,167.315,53.291,159.865
C01534=1017.260,158.086,378.300,167.319,53.282,159.864
C01535=1017.265,158.335,378.280,167.323,53.273,159.863
C01536=1017.270,158.584,378.260,167.325,53.263,159.862
C01537=1017.274,158.834,378.239,167.330,53.254,159.861
C01538=1017.278,159.083,378.219,167.333,53.245,159.859
C01539=1017.283,159.332,378.198,167.336,53.236,159.858
C01540=1017.287,159.581,378.177,167.340,53.226,159.857
C01541=1017.293,159.830,378.157,167.343,53.218,159.856
C01542=1017.297,160.079,378.135,167.348,53.209,159.855
C01543=1017.302,160.328,378.115,167.351,53.200,159.854
C01544=1017.306,160.577,378.094,167.355,53.191,159.853
C01545=1017.311,160.826,378.073,167.358,53.182,159.852
C01546=1017.315,161.075,378.053,167.361,53.173,159.851
C01547=1017.320,161.324,378.032,167.365,53.163,159.850
C01548=1017.325,161.573,378.011,167.368,53.155,159.849
C01549=1017.329,161.822,377.990,167.372,53.145,159.848
C01550=1017.334,162.072,377.969,167.376,53.136,159.846
C01551=1017.339,162.321,377.949,167.380,53.127,159.845
C01552=1017.343,162.569,377.928,167.383,53.118,159.844
C01553=1017.348,162.819,377.907,167.387,53.109,159.843
C01554=1017.353,163.068,377.886,167.390,53.100,159.842
C01555=1017.357,163.317,377.865,167.394,53.091,159.841
C01556=1017.362,163.566,377.845,167.397,53.082,159.840
C01557=1017.366,163.815,377.824,167.401,53.072,159.839
C01558=1017.372,164.064,377.803,167.405,53.064,159.838
C01559=1017.375,164.313,377.782,167.409,53.054,159.837
C01560=1017.381,164.562,377.762,167.412,53.045,159.835
C01561=1017.385,164.812,377.741,167.416,53.036,159.834
C01562=1017.389,165.060,377.720,167.419,53.027,159.833
C01563=1017.394,165.310,377.699,167.423,53.018,159.832
C01564=1017.399,165.559,377.678,167.427,53.009,159.831
C01565=1017.404,165.808,377.658,167.431,53.000,159.830
C01566=1017.408,166.057,377.637,167.435,52.991,159.829
C01567=1017.413,166.306,377.616,167.438,52.982,159.828
C01568=1017.418,166.555,377.594,167.442,52.972,159.827
C01569=1017.423,166.804,377.573,167.445,52.964,159.826
C01570=1017.428,167.053,377.553,167.450,52.954,159.825
C01571=1017.432,167.302,377.532,167.453,52.945,159.823
C01572=1017.436,167.552,377.511,167.457,52.936,159.822
C01573=1017.442,167.801,377.490,167.461,52.927,159.821
C01574=1017.446,168.050,377.469,167.464,52.918,159.820
C01575=1017.452,168.299,377.448,167.468,52.909,159.819
C01576=1017.456,168.547,377.427,167.471,52.899,159.818
C01577=1017.460,168.797,377.406,167.475,52.890,159.817
C01578=1017.465,169.046,377.385,167.478,52.881,159.815
C01579=1017.470,169.295,377.364,167.483,52.872,159.814
C01580=1017.475,169.544,377.342,167.487,52.863,159.813
C01581=1017.480,169.793,377.322,167.490,52.854,159.812
C01582=1017.484,170.042,377.301,167.494,52.844,159.811
C01583=1017.489,170.291,377.280,167.498,52.835,159.810
C01584=1017.494,170.540,377.259,167.502,52.826,159.809
C01585=1017.499,170.821,377.235,167.506,52.816,159.808
C01586=1017.504,171.103,377.211,167.510,52.806,159.807
C01587=1017.511,171.383,377.188,167.515,52.796,159.806
C01588=1017.516,171.664,377.164,167.519,52.785,159.804
C01589=1017.520,171.914,377.143,167.523,52.776,159.803
C01590=1017.525,172.162,377.121,167.527,52.767,159.802
C01591=1017.531,172.412,377.100,167.531,52.758,159.801
C01592=1017.535,172.661,377.079,167.534,52.749,159.800
C01593=1017.541,172.909,377.058,167.538,52.740,159.799
C01594=1017.545,173.158,377.037,167.543,52.730,159.798
C01595=1017.549,173.408,377.016,167.546,52.721,159.797
C01596=1017.555,173.656,376.995,167.550,52.712,159.796
C01597=1017.559,173.906,376.974,167.554,52.703,159.794
C01598=1017.564,174.155,376.953,167.557,52.694,159.793
C01599=1017.569,174.404,376.931,167.562,52.685,159.792
C01600=1017.574,174.653,376.910,167.566,52.676,159.791
C01601=1017.579,174.901,376.889,167.570,52.667,159.790
C01602=1017.584,175.151,376.868,167.573,52.658,159.789
C01603=1017.588,175.400,376.846,167.578,52.649,159.788
C01604=1017.594,175.649,376.825,167.582,52.639,159.787
C01605=1017.598,175.898,376.804,167.585,52.631,159.786
C01606=1017.604,176.147,376.783,167.589,52.621,159.785
C01607=1017.608,176.396,376.762,167.593,52.611,159.784
C01608=1017.613,176.645,376.740,167.597,52.602,159.783
C01609=1017.619,176.894,376.719,167.601,52.593,159.781
C01610=1017.623,177.143,376.697,167.605,52.584,159.780
C01611=1017.628,177.392,376.676,167.609,52.575,159.779
C01612=1017.633,177.641,376.655,167.613,52.566,159.778
C01613=1017.638,177.890,376.634,167.617,52.557,159.777
C01614=1017.644,178.139,376.613,167.621,52.548,159.776
C01615=1017.648,178.388,376.591,167.625,52.539,159.775
C01616=1017.653,178.638,376.569,167.629,52.530,159.774
C01617=1017.659,178.887,376.549,167.634,52.520,159.773
C01618=1017.664,179.136,376.527,167.637,52.512,159.772
C01619=1017.668,179.385,376.506,167.641,52.502,159.771
C01620=1017.674,179.634,376.484,167.646,52.493,159.770
C01621=1017.678,179.882,376.462,167.650,52.484,159.769
C01622=1017.684,180.132,376.442,167.654,52.475,159.768
C01623=1017.689,180.380,376.420,167.657,52.466,159.767
C01624=1017.693,180.630,376.399,167.662,52.457,159.766
C01625=1017.699,180.878,376.378,167.665,52.447,159.764
C01626=1017.704,181.128,376.355,167.670,52.438,159.763
C01627=1017.709,181.377,376.334,167.674,52.429,159.762
C01628=1017.714,181.626,376.313,167.677,52.420,159.761
C01629=1017.719,181.875,376.292,167.682,52.411,159.760
C01630=1017.723,182.124,376.270,167.686,52.402,159.759
C01631=1017.728,182.373,376.248,167.691,52.393,159.758
C01632=1017.733,182.623,376.225,167.694,52.385,159.757
C01633=1017.738,182.872,376.203,167.698,52.375,159.756
C01634=1017.742,183.121,376.181,167.702,52.367,159.755
C01635=1017.747,183.369,376.159,167.706,52.358,159.754
C01636=1017.752,183.618,376.137,167.710,52.349,159.753
C01637=1017.756,183.867,376.115,167.714,52.340,159.752
C01638=1017.760,184.116,376.093,167.719,52.332,159.751
C01639=1017.765,184.365,376.071,167.723,52.323,159.750
C01640=1017.771,184.615,376.049,167.727,52.314,159.749
C01641=1017.776,184.863,376.027,167.731,52.305,159.748
C01642=1017.780,185.113,376.004,167.735,52.296,159.747
C01643=1017.784,185.361,375.983,167.739,52.287,159.746
C01644=1017.789,185.610,375.961,167.743,52.278,159.745
C01645=1017.794,185.859,375.938,167.748,52.270,159.744
C01646=1017.799,186.108,375.915,167.752,52.261,159.743
C01647=1017.804,186.357,375.893,167.755,52.252,159.742
C01648=1017.809,186.606,375.872,167.760,52.244,159.741
C01649=1017.814,186.887,375.847,167.765,52.234,159.740
C01650=1017.819,187.167,375.822,167.770,52.223,159.739
C01651=1017.824,187.448,375.797,167.774,52.214,159.737
C01652=1017.830,187.728,375.772,167.779,52.203,159.736
C01653=1017.835,187.978,375.749,167.783,52.195,159.736
C01654=1017.839,188.226,375.727,167.788,52.186,159.735
C01655=1017.844,188.475,375.705,167.791,52.177,159.733
C01656=1017.849,188.724,375.682,167.795,52.168,159.732
C01657=1017.854,188.973,375.660,167.800,52.160,159.732
C01658=1017.859,189.222,375.638,167.804,52.151,159.730
C01659=1017.864,189.471,375.616,167.808,52.142,159.729
C01660=1017.868,189.719,375.593,167.812,52.133,159.728
C01661=1017.874,189.969,375.571,167.817,52.124,159.727
C01662=1017.878,190.218,375.549,167.821,52.115,159.726
C01663=1017.883,190.467,375.526,167.826,52.106,159.725
C01664=1017.888,190.716,375.503,167.829,52.098,159.724
C01665=1017.893,190.965,375.481,167.834,52.089,159.723
C01666=1017.897,191.214,375.459,167.838,52.080,159.722
C01667=1017.903,191.463,375.436,167.842,52.071,159.721
C01668=1017.908,191.711,375.414,167.847,52.063,159.721
C01669=1017.913,191.960,375.392,167.850,52.054,159.719
C01670=1017.917,192.210,375.369,167.855,52.045,159.718
C01671=1017.922,192.458,375.347,167.860,52.036,159.718
C01672=1017.927,192.707,375.325,167.864,52.027,159.717
C01673=1017.932,192.956,375.302,167.868,52.018,159.716
C01674=1017.937,193.205,375.280,167.873,52.009,159.714
C01675=1017.942,193.454,375.258,167.878,52.001,159.714
C01676=1017.947,193.703,375.234,167.881,51.992,159.713
C01677=1017.952,193.952,375.212,167.885,51.983,159.711
C01678=1017.957,194.201,375.189,167.890,51.975,159.711
C01679=1017.962,194.450,375.168,167.894,51.966,159.710
C01680=1017.966,194.699,375.145,167.899,51.956,159.709
C01681=1017.972,194.948,375.122,167.904,51.948,159.708
C01682=1017.977,195.196,375.100,167.908,51.939,159.707
C01683=1017.982,195.446,375.077,167.912,51.930,159.706
C01684=1017.987,195.695,375.055,167.917,51.921,159.705
C01685=1017.992,195.943,375.032,167.921,51.913,159.704
C01686=1017.996,196.193,375.009,167.925,51.904,159.703
C01687=1018.002,196.441,374.987,167.929,51.895,159.702
C01688=1018.007,196.690,374.965,167.934,51.887,159.701
C01689=1018.012,196.939,374.941,167.939,51.877,159.700
C01690=1018.017,197.188,374.919,167.943,51.868,159.699
C01691=1018.023,197.437,374.896,167.948,51.860,159.698
C01692=1018.027,197.686,374.874,167.952,51.851,159.697
C01693=1018.032,197.935,374.851,167.957,51.842,159.696
C01694=1018.037,198.183,374.828,167.961,51.834,159.695
C01695=1018.042,198.433,374.806,167.966,51.825,159.694
C01696=1018.047,198.681,374.783,167.970,51.816,159.693
C01697=1018.053,198.931,374.761,167.975,51.807,159.692
C01698=1018.058,199.179,374.738,167.979,51.798,159.691
C01699=1018.063,199.428,374.715,167.984,51.789,159.690
C01700=1018.067,199.677,374.692,167.989,51.781,159.689
C01701=1018.073,199.926,374.669,167.992,51.772,159.688
C01702=1018.077,200.175,374.646,167.997,51.764,159.687
C01703=1018.082,200.424,374.622,168.001,51.755,159.686
C01704=1018.088,200.673,374.600,168.006,51.747,159.685
C01705=1018.092,200.921,374.576,168.011,51.738,159.684
C01706=1018.097,201.171,374.554,168.015,51.729,159.684
C01707=1018.101,201.420,374.530,168.020,51.720,159.683
C01708=1018.107,201.669,374.507,168.025,51.712,159.682
C01709=1018.111,201.917,374.484,168.029,51.703,159.681
C01710=1018.116,202.166,374.461,168.034,51.695,159.680
C01711=1018.122,202.415,374.438,168.038,51.686,159.679
C01712=1018.126,202.664,374.415,168.042,51.678,159.678
C01713=1018.152,203.903,374.298,168.519,51.768,159.786
C01714=1018.158,204.134,374.275,168.522,51.761,159.786
C01715=1018.163,204.366,374.252,168.526,51.754,159.785
C01716=1018.168,204.597,374.229,168.529,51.747,159.784
C01717=1018.175,204.828,374.206,168.532,51.740,159.783
C01718=1018.180,205.059,374.183,168.536,51.733,159.782
C01719=1018.185,205.290,374.160,168.540,51.726,159.781
C01720=1018.191,205.522,374.137,168.544,51.719,159.781
C01721=1018.197,205.771,374.111,168.548,51.712,159.780
C01722=1018.203,206.019,374.086,168.551,51.704,159.779
C01723=1018.209,206.268,374.062,168.555,51.697,159.778
C01724=1018.215,206.517,374.037,168.559,51.689,159.777
C01725=1018.220,206.765,374.012,168.563,51.682,159.776
C01726=1018.226,207.014,373.987,168.567,51.674,159.775
C01727=1018.233,207.263,373.962,168.571,51.666,159.774
C01728=1018.238,207.511,373.937,168.575,51.659,159.774
C01729=1018.244,207.760,373.912,168.578,51.652,159.773
C01730=1018.250,208.009,373.887,168.582,51.644,159.772
C01731=1018.256,208.257,373.862,168.586,51.637,159.771
C01732=1018.261,208.506,373.836,168.590,51.630,159.770
C01733=1018.267,208.755,373.811,168.595,51.623,159.769
C01734=1018.274,209.004,373.786,168.597,51.615,159.768
C01735=1018.279,209.252,373.762,168.601,51.608,159.768
C01736=1018.285,209.501,373.736,168.606,51.601,159.767
C01737=1018.291,209.749,373.711,168.610,51.593,159.766
C01738=1018.298,209.998,373.686,168.614,51.585,159.765
C01739=1018.303,210.246,373.661,168.617,51.579,159.764
C01740=1018.309,210.495,373.635,168.621,51.571,159.763
C01741=1018.314,210.744,373.610,168.625,51.564,159.763
C01742=1018.321,210.993,373.585,168.629,51.557,159.762
C01743=1018.326,211.241,373.559,168.633,51.550,159.761
C01744=1018.332,211.490,373.534,168.637,51.543,159.760
C01745=1018.338,211.739,373.508,168.641,51.536,159.759
C01746=1018.344,211.987,373.483,168.645,51.528,159.759
C01747=1018.349,212.236,373.458,168.648,51.522,159.758
C01748=1018.355,212.484,373.432,168.652,51.514,159.757
C01749=1018.361,212.733,373.407,168.656,51.506,159.756
C01750=1018.368,212.982,373.382,168.660,51.500,159.755
C01751=1018.373,213.231,373.356,168.664,51.492,159.754
C01752=1018.379,213.479,373.330,168.668,51.485,159.753
C01753=1018.385,213.727,373.305,168.672,51.478,159.753
C01754=1018.390,213.976,373.279,168.675,51.471,159.752
C01755=1018.397,214.225,373.254,168.680,51.464,159.751
C01756=1018.403,214.474,373.229,168.684,51.457,159.750
C01757=1018.409,214.722,373.203,168.688,51.449,159.749
C01758=1018.414,214.971,373.177,168.692,51.443,159.749
C01759=1018.421,215.220,373.152,168.696,51.436,159.748
C01760=1018.426,215.468,373.127,168.700,51.429,159.747
C01761=1018.433,215.717,373.102,168.703,51.422,159.746
C01762=1018.438,215.965,373.076,168.708,51.415,159.746
C01763=1018.444,216.214,373.050,168.712,51.408,159.745
C01764=1018.450,216.463,373.025,168.715,51.401,159.744
C01765=1018.456,216.712,372.999,168.719,51.394,159.743
C01766=1018.462,216.960,372.973,168.724,51.386,159.742
C01767=1018.469,217.209,372.948,168.728,51.379,159.742
C01768=1018.474,217.458,372.922,168.731,51.373,159.741
C01769=1018.480,217.706,372.897,168.736,51.366,159.740
C01770=1018.486,217.954,372.872,168.740,51.359,159.739
C01771=1018.492,218.202,372.846,168.743,51.352,159.738
C01772=1018.498,218.451,372.820,168.747,51.345,159.738
C01773=1018.503,218.682,372.796,168.751,51.339,159.737
C01774=1018.509,218.912,372.771,168.755,51.332,159.736
C01775=1018.514,219.142,372.747,168.758,51.326,159.736
C01776=1018.519,219.373,372.724,168.762,51.320,159.735
C01777=1018.525,219.603,372.699,168.765,51.314,159.734
C01778=1018.531,219.832,372.676,168.770,51.307,159.734
C01779=1018.536,220.062,372.652,168.773,51.301,159.733
C01780=1018.542,220.293,372.628,168.777,51.294,159.732
C01781=1018.547,220.542,372.602,168.781,51.288,159.732
C01782=1018.554,220.790,372.576,168.785,51.281,159.731
C01783=1018.559,221.039,372.550,168.788,51.275,159.730
C01784=1018.565,221.287,372.524,168.793,51.268,159.729
C01785=1018.571,221.536,372.498,168.797,51.261,159.729
C01786=1018.576,221.785,372.472,168.801,51.254,159.728
C01787=1018.583,222.033,372.446,168.805,51.247,159.727
C01788=1018.588,222.282,372.420,168.809,51.241,159.726
C01789=1018.594,222.530,372.394,168.813,51.234,159.726
C01790=1018.600,222.779,372.368,168.817,51.228,159.725
C01791=1018.606,223.027,372.342,168.821,51.221,159.724
C01792=1018.612,223.276,372.316,168.825,51.214,159.724
C01793=1018.618,223.524,372.290,168.829,51.207,159.723
C01794=1018.624,223.773,372.264,168.833,51.201,159.722
C01795=1018.631,224.022,372.237,168.836,51.194,159.721
C01796=1018.636,224.271,372.211,168.841,51.188,159.721
C01797=1018.643,224.519,372.185,168.846,51.181,159.720
C01798=1018.648,224.768,372.159,168.849,51.174,159.719
C01799=1018.655,225.016,372.133,168.854,51.168,159.719
C01800=1018.660,225.265,372.107,168.857,51.161,159.718
C01801=1018.666,225.513,372.081,168.862,51.155,159.717
C01802=1018.672,225.761,372.055,168.865,51.148,159.716
C01803=1018.678,226.010,372.029,168.870,51.141,159.716
C01804=1018.684,226.258,372.003,168.873,51.135,159.715
C01805=1018.690,226.508,371.976,168.877,51.128,159.714
C01806=1018.696,226.756,371.950,168.881,51.122,159.714
C01807=1018.702,227.005,371.923,168.886,51.115,159.713
C01808=1018.709,227.253,371.897,168.889,51.109,159.712
C01809=1018.714,227.502,371.871,168.894,51.102,159.712
C01810=1018.720,227.750,371.844,168.897,51.096,159.711
C01811=1018.726,227.998,371.818,168.902,51.090,159.710
C01812=1018.731,228.247,371.791,168.906,51.083,159.710
C01813=1018.738,228.496,371.764,168.910,51.077,159.709
C01814=1018.743,228.745,371.738,168.914,51.071,159.709
C01815=1018.750,228.993,371.712,168.918,51.064,159.708
C01816=1018.755,229.241,371.686,168.922,51.058,159.707
C01817=1018.761,229.490,371.659,168.927,51.051,159.706
C01818=1018.767,229.738,371.632,168.930,51.045,159.706
C01819=1018.773,229.987,371.605,168.935,51.039,159.705
C01820=1018.779,230.235,371.579,168.939,51.033,159.705
C01821=1018.785,230.484,371.552,168.942,51.026,159.704
C01822=1018.791,230.732,371.525,168.947,51.020,159.703
